FUNCTION "Take-up unit" : VOID	// FC 7
TITLE = TAKE-UP UNIT FUNCTION
AUTHOR : Milesi
VERSION : 0.1
VAR_TEMP
  Min_diameter : REAL ;
  T_up_linear_speed : REAL ;
  T_up_speed_ref : REAL ;
  Take_up_speed_ref : REAL ;
END_VAR
BEGIN
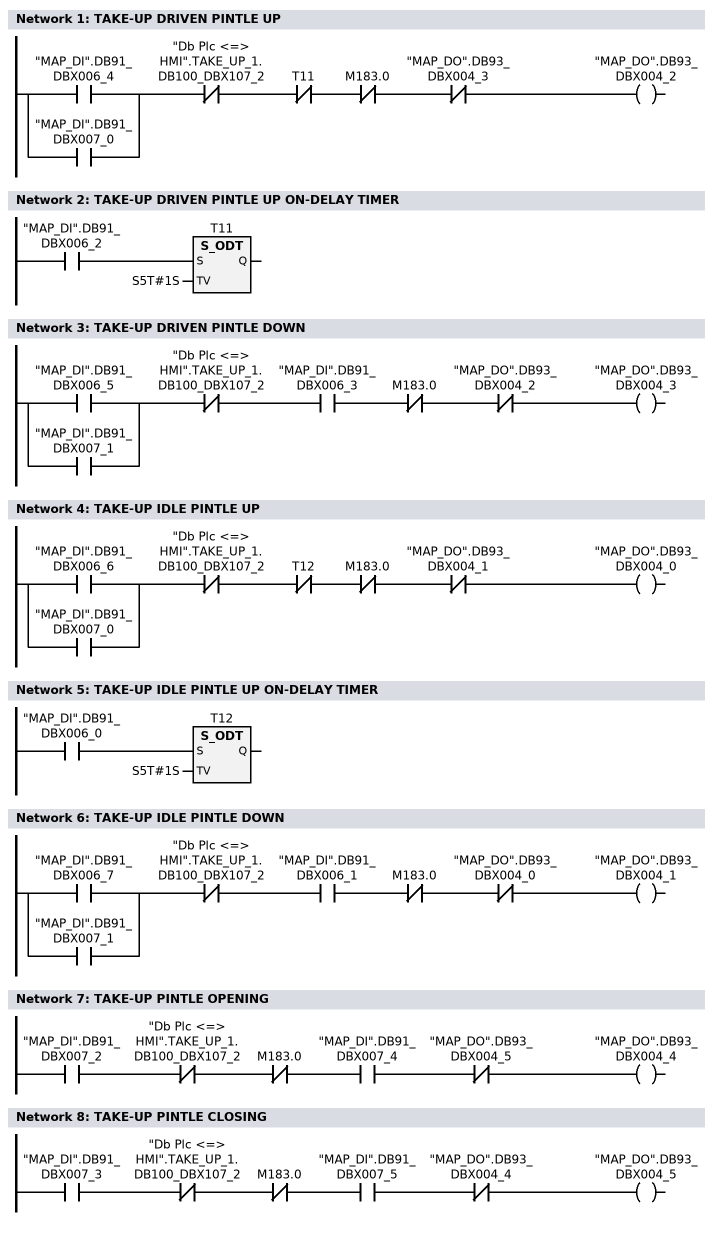
NETWORK
TITLE = TAKE-UP DRIVEN PINTLE UP
      A(;
      O     "MAP_DI".DB91_DBX006_4;
      O     "MAP_DI".DB91_DBX007_0;
      );
      AN    "Db Plc <=> HMI".TAKE_UP_1.DB100_DBX107_2;
      AN    "T11";
      AN    "M183.0";
      AN    "MAP_DO".DB93_DBX004_3;
      =     "MAP_DO".DB93_DBX004_2;
NETWORK
TITLE = TAKE-UP DRIVEN PINTLE UP ON-DELAY TIMER
      A     "MAP_DI".DB91_DBX006_2;
      L     S5T#1S;
      SD    "T11";
      NOP   0;
      NOP   0;
      NOP   0;
      NOP   0;
NETWORK
TITLE = TAKE-UP DRIVEN PINTLE DOWN
      A(;
      O     "MAP_DI".DB91_DBX006_5;
      O     "MAP_DI".DB91_DBX007_1;
      );
      AN    "Db Plc <=> HMI".TAKE_UP_1.DB100_DBX107_2;
      A     "MAP_DI".DB91_DBX006_3;
      AN    "M183.0";
      AN    "MAP_DO".DB93_DBX004_2;
      =     "MAP_DO".DB93_DBX004_3;
NETWORK
TITLE = TAKE-UP IDLE PINTLE UP
      A(;
      O     "MAP_DI".DB91_DBX006_6;
      O     "MAP_DI".DB91_DBX007_0;
      );
      AN    "Db Plc <=> HMI".TAKE_UP_1.DB100_DBX107_2;
      AN    "T12";
      AN    "M183.0";
      AN    "MAP_DO".DB93_DBX004_1;
      =     "MAP_DO".DB93_DBX004_0;
NETWORK
TITLE = TAKE-UP IDLE PINTLE UP ON-DELAY TIMER
      A     "MAP_DI".DB91_DBX006_0;
      L     S5T#1S;
      SD    "T12";
      NOP   0;
      NOP   0;
      NOP   0;
      NOP   0;
NETWORK
TITLE = TAKE-UP IDLE PINTLE DOWN
      A(;
      O     "MAP_DI".DB91_DBX006_7;
      O     "MAP_DI".DB91_DBX007_1;
      );
      AN    "Db Plc <=> HMI".TAKE_UP_1.DB100_DBX107_2;
      A     "MAP_DI".DB91_DBX006_1;
      AN    "M183.0";
      AN    "MAP_DO".DB93_DBX004_0;
      =     "MAP_DO".DB93_DBX004_1;
NETWORK
TITLE = TAKE-UP PINTLE OPENING
      A     "MAP_DI".DB91_DBX007_2;
      AN    "Db Plc <=> HMI".TAKE_UP_1.DB100_DBX107_2;
      AN    "M183.0";
      A     "MAP_DI".DB91_DBX007_4;
      AN    "MAP_DO".DB93_DBX004_5;
      =     "MAP_DO".DB93_DBX004_4;
NETWORK
TITLE = TAKE-UP PINTLE CLOSING
      A     "MAP_DI".DB91_DBX007_3;
      AN    "Db Plc <=> HMI".TAKE_UP_1.DB100_DBX107_2;
      AN    "M183.0";
      A     "MAP_DI".DB91_DBX007_5;
      AN    "MAP_DO".DB93_DBX004_4;
      =     "MAP_DO".DB93_DBX004_5;
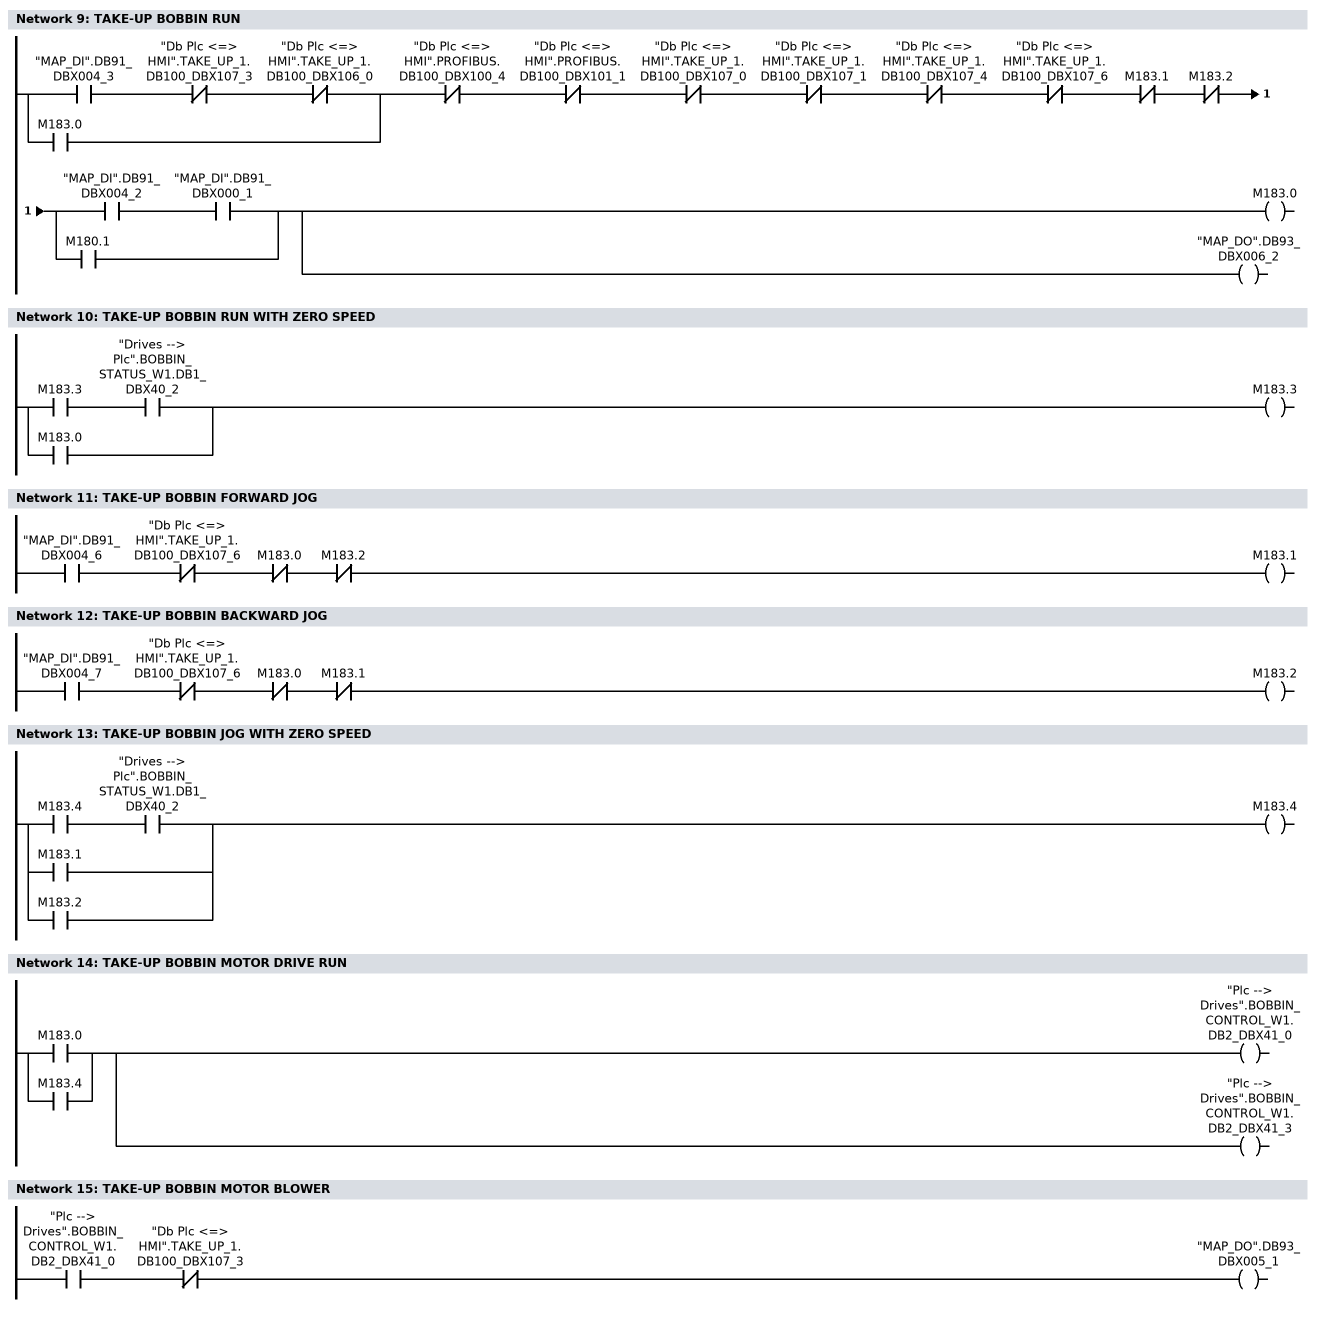
NETWORK
TITLE = TAKE-UP BOBBIN RUN
      A(;
      A     "MAP_DI".DB91_DBX004_3;
      AN    "Db Plc <=> HMI".TAKE_UP_1.DB100_DBX107_3;
      AN    "Db Plc <=> HMI".TAKE_UP_1.DB100_DBX106_0;
      O     "M183.0";
      );
      AN    "Db Plc <=> HMI".PROFIBUS.DB100_DBX100_4;
      AN    "Db Plc <=> HMI".PROFIBUS.DB100_DBX101_1;
      AN    "Db Plc <=> HMI".TAKE_UP_1.DB100_DBX107_0;
      AN    "Db Plc <=> HMI".TAKE_UP_1.DB100_DBX107_1;
      AN    "Db Plc <=> HMI".TAKE_UP_1.DB100_DBX107_4;
      AN    "Db Plc <=> HMI".TAKE_UP_1.DB100_DBX107_6;
      AN    "M183.1";
      AN    "M183.2";
      A(;
      A     "MAP_DI".DB91_DBX004_2;
      A     "MAP_DI".DB91_DBX000_1;
      O     "M180.1";
      );
      =     "M183.0";
      =     "MAP_DO".DB93_DBX006_2;
NETWORK
TITLE = TAKE-UP BOBBIN RUN WITH ZERO SPEED
      A     "M183.3";
      A     "Drives --> Plc".BOBBIN_STATUS_W1.DB1_DBX40_2;
      O     "M183.0";
      =     "M183.3";
NETWORK
TITLE = TAKE-UP BOBBIN FORWARD JOG
      A     "MAP_DI".DB91_DBX004_6;
      AN    "Db Plc <=> HMI".TAKE_UP_1.DB100_DBX107_6;
      AN    "M183.0";
      AN    "M183.2";
      =     "M183.1";
NETWORK
TITLE = TAKE-UP BOBBIN BACKWARD JOG
      A     "MAP_DI".DB91_DBX004_7;
      AN    "Db Plc <=> HMI".TAKE_UP_1.DB100_DBX107_6;
      AN    "M183.0";
      AN    "M183.1";
      =     "M183.2";
NETWORK
TITLE = TAKE-UP BOBBIN JOG WITH ZERO SPEED
      A     "M183.4";
      A     "Drives --> Plc".BOBBIN_STATUS_W1.DB1_DBX40_2;
      O     "M183.1";
      O     "M183.2";
      =     "M183.4";
NETWORK
TITLE = TAKE-UP BOBBIN MOTOR DRIVE RUN
      O     "M183.0";
      O     "M183.4";
      =     "Plc --> Drives".BOBBIN_CONTROL_W1.DB2_DBX41_0;
      =     "Plc --> Drives".BOBBIN_CONTROL_W1.DB2_DBX41_3;
NETWORK
TITLE = TAKE-UP BOBBIN MOTOR BLOWER
      A     "Plc --> Drives".BOBBIN_CONTROL_W1.DB2_DBX41_0;
      AN    "Db Plc <=> HMI".TAKE_UP_1.DB100_DBX107_3;
      =     "MAP_DO".DB93_DBX005_1;
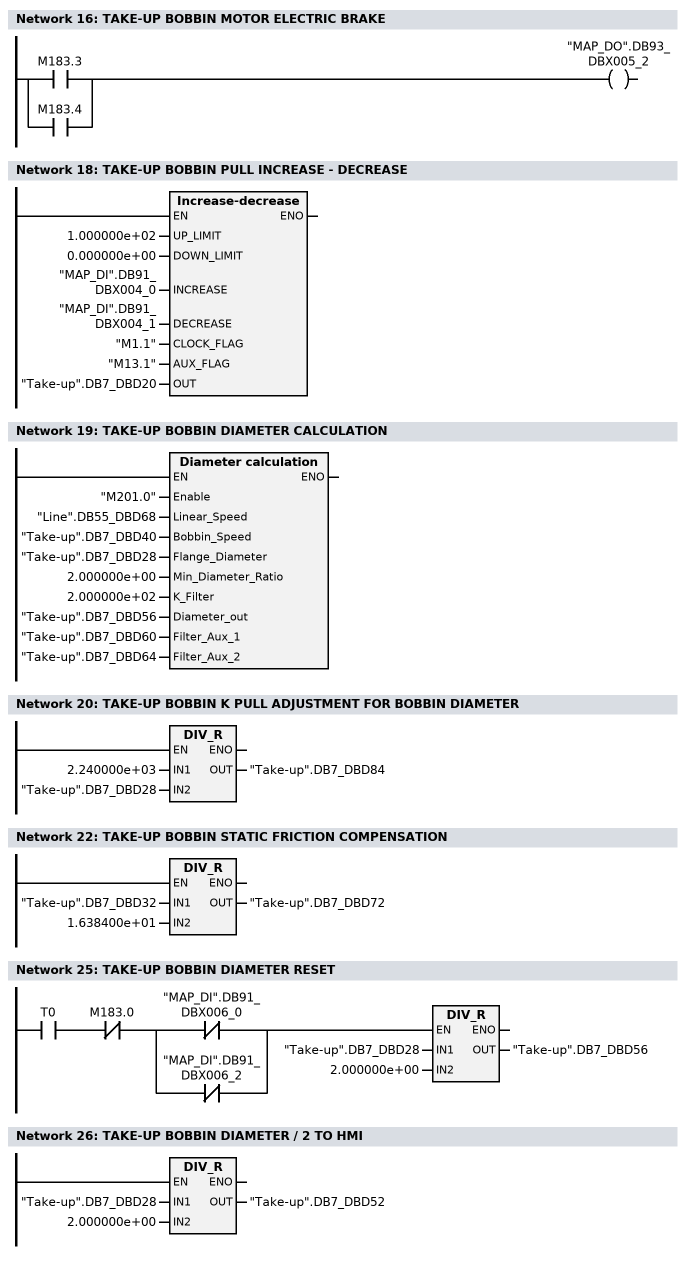
NETWORK
TITLE = TAKE-UP BOBBIN MOTOR ELECTRIC BRAKE
      O     "M183.3";
      O     "M183.4";
      =     "MAP_DO".DB93_DBX005_2;
NETWORK
TITLE = TAKE-UP BOBBIN RPM
      L     "Drives --> Plc".DB1_DBW46;
      ITD;
      DTR;
      L     1.638400e+04;
      /R;
      L     3.031000e+01;
      *R;
      ABS;
      T     "Take-up".DB7_DBD40;
NETWORK
TITLE = TAKE-UP BOBBIN PULL INCREASE - DECREASE
      CALL  "Increase-decrease" (
           UP_LIMIT                 := 1.000000e+02,
           DOWN_LIMIT               := 0.000000e+00,
           INCREASE                 := "MAP_DI".DB91_DBX004_0,
           DECREASE                 := "MAP_DI".DB91_DBX004_1,
           CLOCK_FLAG               := "M1.1",
           AUX_FLAG                 := "M13.1",
           OUT                      := "Take-up".DB7_DBD20);
NETWORK
TITLE = TAKE-UP BOBBIN DIAMETER CALCULATION
      CALL  "Diameter calculation" (
           Enable                   := "M201.0",
           Linear_Speed             := "Line".DB55_DBD68,
           Bobbin_Speed             := "Take-up".DB7_DBD40,
           Flange_Diameter          := "Take-up".DB7_DBD28,
           Min_Diameter_Ratio       := 2.000000e+00,
           K_Filter                 := 2.000000e+02,
           Diameter_out             := "Take-up".DB7_DBD56,
           Filter_Aux_1             := "Take-up".DB7_DBD60,
           Filter_Aux_2             := "Take-up".DB7_DBD64);
NETWORK
TITLE = TAKE-UP BOBBIN K PULL ADJUSTMENT FOR BOBBIN DIAMETER 
      L     2.240000e+03;
      L     "Take-up".DB7_DBD28;
      /R;
      T     "Take-up".DB7_DBD84;
NETWORK
TITLE = TAKE-UP BOBBIN PULL REFERENCE
//Max diameter bobbin = 2240
//Max pull set = 100
//
//(Max diameter bobbin * Max pull set)
//------------------------------------ = 16384
//                 K
//
//    (Max diameter bobbin * Max pull set)   2240 * 100
//K = ------------------------------------ = ---------- = 13.67187
//                    16384                    16384
      L     "Take-up".DB7_DBD56;
      L     "Take-up".DB7_DBD20;
      *R;
      L     1.367187e+01;
      /R;
      L     "Take-up".DB7_DBD84;
      *R;
      L     "Take-up".DB7_DBD72;
      +R;
      L     "Take-up".DB7_DBD76;
      +R;
      T     "Take-up".DB7_DBD68;
NETWORK
TITLE = TAKE-UP BOBBIN STATIC FRICTION COMPENSATION
      L     "Take-up".DB7_DBD32;
      L     1.638400e+01;
      /R;
      T     "Take-up".DB7_DBD72;
NETWORK
TITLE = TAKE-UP BOBBIN DYNAMIC FRICTION COMPENSATION
//Max Bobbin rpm = 30.31
//Max dynamic friction set = 100
//
//(Max Bobbin rpm * Max dynamic friction set) * K = 1638
//
//              1638                                   1638 
//K = ------------------------------------------- = ----------- = 0.54041
//    (Max Bobbin rpm * Max dynamic friction set)   30.31 * 100
      L     "Take-up".DB7_DBD40;
      L     "Take-up".DB7_DBD36;
      *R;
      L     5.404100e-01;
      /R;
      T     "Take-up".DB7_DBD76;
NETWORK
TITLE = TAKE-UP BOBBIN MINIMUM PULL WITH LINE STOP
      A     "M180.1";
      JC    _032;
      L     "Take-up".DB7_DBD56;
      L     "Take-up".DB7_DBD20;
      *R;
      L     1.367187e+01;
      /R;
      L     "Take-up".DB7_DBD24;
      *R;
      L     1.000000e+02;
      /R;
      L     "Take-up".DB7_DBD72;
      +R;
      T     "Take-up".DB7_DBD68;
_032: NOP   0;
NETWORK
TITLE = TAKE-UP BOBBIN DIAMETER RESET
      A     "T0";
      AN    "M183.0";
      A(;
      ON    "MAP_DI".DB91_DBX006_0;
      ON    "MAP_DI".DB91_DBX006_2;
      );
      JNB   _001;
      L     "Take-up".DB7_DBD28;
      L     2.000000e+00;
      /R;
      T     "Take-up".DB7_DBD56;
_001: NOP   0;
NETWORK
TITLE = TAKE-UP BOBBIN DIAMETER / 2 TO HMI
      L     "Take-up".DB7_DBD28;
      L     2.000000e+00;
      /R;
      T     "Take-up".DB7_DBD52;
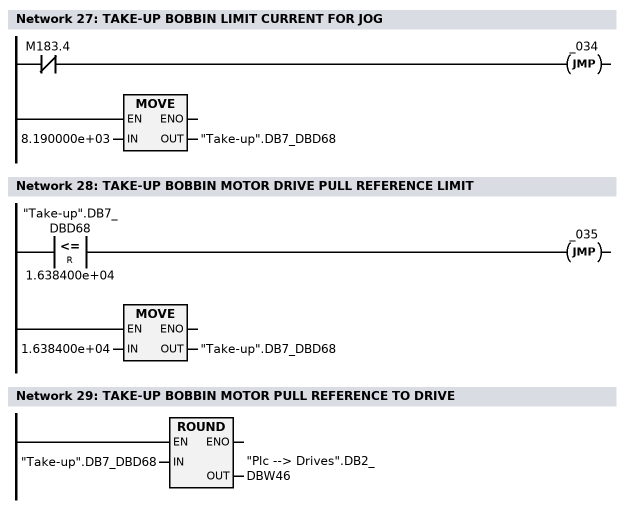
NETWORK
TITLE = TAKE-UP BOBBIN LIMIT CURRENT FOR JOG
      AN    "M183.4";
      JC    _034;
      L     8.190000e+03;
      T     "Take-up".DB7_DBD68;
_034: NOP   0;
NETWORK
TITLE = TAKE-UP BOBBIN MOTOR DRIVE PULL REFERENCE LIMIT
      A(;
      L     "Take-up".DB7_DBD68;
      L     1.638400e+04;
      <=R;
      );
      JC    _035;
      L     1.638400e+04;
      T     "Take-up".DB7_DBD68;
_035: NOP   0;
NETWORK
TITLE = TAKE-UP BOBBIN MOTOR PULL REFERENCE TO DRIVE
      L     "Take-up".DB7_DBD68;
      RND;
      T     "Plc --> Drives".DB2_DBW46;
NETWORK
TITLE = TAKE-UP BOBBIN MOTOR SPEED REFERENCE TO DRIVE
// (network holds code this reader does not know; not shown)
NETWORK
TITLE = TAKE-UP BOBBIN MOTOR RPM TO HMI
      L     "Drives --> Plc".DB1_DBW46;
      ITD;
      DTR;
      L     1.638400e+04;
      /R;
      L     1.515000e+03;
      *R;
      T     "Take-up".DB7_DBD188;
NETWORK
TITLE = TAKE-UP BOBBIN MOTOR CURRENT TO HMI
      L     "Drives --> Plc".DB1_DBW48;
      ITD;
      DTR;
      L     1.638400e+04;
      /R;
      L     2.150000e+01;
      *R;
      T     "Take-up".DB7_DBD192;
NETWORK
TITLE = TAKE-UP BOBBIN MOTOR VOLTAGE TO HMI
      L     "Drives --> Plc".DB1_DBW50;
      ITD;
      DTR;
      L     1.638400e+04;
      /R;
      L     4.000000e+02;
      *R;
      T     "Take-up".DB7_DBD196;
END_FUNCTION

FUNCTION "Capstan alarms" : VOID	// FC 8
TITLE = CAPSTAN ALARMS FUNCTION
AUTHOR : Milesi
VERSION : 0.1
BEGIN
NETWORK
TITLE = CAPSTAN MOTOR DRIVE PROFIBUS SLAVE 5 FAULT
      A(;
      L     "MB304";
      L     5;
      ==I;
      );
      AN    "M300.5";
      S     "Db Plc <=> HMI".PROFIBUS.DB100_DBX101_2;
NETWORK
TITLE = CAPSTAN MOTOR DRIVE FAULT
      A     "T0";
      A     "Drives --> Plc".CAPSTAN_STATUS_W1.DB1_DBX81_3;
      S     "Db Plc <=> HMI".CAPSTAN.DB100_DBX109_6;
NETWORK
TITLE = CAPSTAN MOTOR OVERTEMPERATURE
      A     "T0";
      A     "Drives --> Plc".CAPSTAN_STATUS_W2.DB1_DBX82_1;
      S     "Db Plc <=> HMI".CAPSTAN.DB100_DBX109_7;
NETWORK
TITLE = CAPSTAN MOTOR BLOWER OVERLOAD
      A     "T0";
      A     "MAP_DI".DB91_DBX012_0;
      =     "Db Plc <=> HMI".CAPSTAN.DB100_DBX109_0;
NETWORK
TITLE = CAPSTAN MOTOR BRAKE CONTROL
      A     "T0";
      A     "M180.1";
      AN    "MAP_DI".DB91_DBX012_2;
      A     "T2";
      S     "Db Plc <=> HMI".CAPSTAN.DB100_DBX109_2;
NETWORK
TITLE = CAPSTAN MAIN AIR MINIMUM PRESSURE
      A     "T0";
      A     "M180.1";
      AN    "MAP_DI".DB91_DBX012_1;
      S     "M170.1";
NETWORK
TITLE =
      A     "T0";
      A(;
      ON    "MAP_DI".DB91_DBX012_1;
      O     "M170.1";
      );
      =     "Db Plc <=> HMI".CAPSTAN.DB100_DBX109_3;
NETWORK
TITLE = CABLE BLOCK OPEN
      A     "T0";
      AN    "M180.1";
      A     "M21.1";
      AN    "M184.0";
      AN    "M184.1";
      A     "MAP_DI".DB91_DBX012_3;
      =     "Db Plc <=> HMI".CAPSTAN.DB100_DBX109_4;
NETWORK
TITLE = CABLE BLOCK CLOSE AFTER RUN
      A     "T0";
      A(;
      O     "M180.1";
      O     "M21.3";
      O     "M184.0";
      O     "M184.1";
      );
      AN    "MAP_DI".DB91_DBX012_3;
      A     "T2";
      S     "Db Plc <=> HMI".CAPSTAN.DB100_DBX109_5;
NETWORK
TITLE = CAPSTAN GENERAL ALARM 
      AN    "Db Plc <=> HMI".PROFIBUS.DB100_DBX101_2;
      AN    "Db Plc <=> HMI".CAPSTAN.DB100_DBX109_0;
      AN    "Db Plc <=> HMI".CAPSTAN.DB100_DBX109_2;
      AN    "Db Plc <=> HMI".CAPSTAN.DB100_DBX109_3;
      AN    "Db Plc <=> HMI".CAPSTAN.DB100_DBX109_4;
      AN    "Db Plc <=> HMI".CAPSTAN.DB100_DBX109_5;
      AN    "Db Plc <=> HMI".CAPSTAN.DB100_DBX109_6;
      AN    "Db Plc <=> HMI".CAPSTAN.DB100_DBX109_7;
      =     "M197.3";
END_FUNCTION

FUNCTION "Capstan unit" : VOID	// FC 9
TITLE = CAPSTAN UNIT FUNCTION
AUTHOR : Milesi
VERSION : 0.1
VAR_TEMP
  Cable_diameter_K : REAL ;
END_VAR
BEGIN
NETWORK
TITLE = CAPSTAN FORWARD JOG
      A     "MAP_DI".DB91_DBX012_5;
      AN    "Db Plc <=> HMI".CAPSTAN.DB100_DBX109_0;
      AN    "Db Plc <=> HMI".CAPSTAN.DB100_DBX109_2;
      AN    "Db Plc <=> HMI".CAPSTAN.DB100_DBX109_5;
      AN    "Db Plc <=> HMI".CAPSTAN.DB100_DBX109_6;
      AN    "Db Plc <=> HMI".CAPSTAN.DB100_DBX109_7;
      AN    "M180.1";
      AN    "M184.1";
      =     "M184.0";
NETWORK
TITLE = CAPSTAN BACKWARD JOG
      A     "MAP_DI".DB91_DBX012_6;
      AN    "Db Plc <=> HMI".CAPSTAN.DB100_DBX109_0;
      AN    "Db Plc <=> HMI".CAPSTAN.DB100_DBX109_2;
      AN    "Db Plc <=> HMI".CAPSTAN.DB100_DBX109_5;
      AN    "Db Plc <=> HMI".CAPSTAN.DB100_DBX109_6;
      AN    "Db Plc <=> HMI".CAPSTAN.DB100_DBX109_7;
      AN    "M180.1";
      AN    "M184.0";
      =     "M184.1";
NETWORK
TITLE = CAPSTAN JOG WITH ZERO SPEED
      A     "M184.2";
      A     "Drives --> Plc".CAPSTAN_STATUS_W1.DB1_DBX80_2;
      O     "M184.0";
      O     "M184.1";
      =     "M184.2";
NETWORK
TITLE = CAPSTAN MOTOR DRIVE RUN
      O     "M21.3";
      O     "M180.1";
      O     "M184.2";
      =     "Plc --> Drives".CAPSTAN_CONTROL_W1.DB2_DBX81_0;
      =     "Plc --> Drives".CAPSTAN_CONTROL_W1.DB2_DBX81_3;
NETWORK
TITLE = CAPSTAN MOTOR BLOWER
      A     "Plc --> Drives".CAPSTAN_CONTROL_W1.DB2_DBX81_0;
      AN    "Db Plc <=> HMI".CAPSTAN.DB100_DBX109_0;
      =     "MAP_DO".DB93_DBX001_2;
NETWORK
TITLE = CAPSTAN BRAKE BLOCK
      A     "M21.1";
      AN    "M180.1";
      AN    "M184.2";
      =     "MAP_DO".DB93_DBX001_3;
NETWORK
TITLE = CAPSTAN CABLE BLOCK
      O     "M180.1";
      O     "M21.3";
      O     "M184.2";
      O;
      A     "MAP_DI".DB91_DBX012_4;
      AN    "M180.1";
      A     "M21.1";
      AN    "M184.2";
      =     "MAP_DO".DB93_DBX001_4;
NETWORK
TITLE = CABLE DIAMETER CONSTANT
//             Capstan pulley Ш + Cable Ш
//K (Cable Ш)= --------------------------
//                 Capstan pulley Ш
      L     2.500000e+03;
      L     "Line".DB55_DBD56;
      +R;
      L     2.500000e+03;
      /R;
      T     #Cable_diameter_K;
NETWORK
TITLE = CAPSTAN MOTOR DRIVE SPEED REFERENCE
// (network holds code this reader does not know; not shown)
NETWORK
TITLE = CAPSTAN MOTOR RPM TO HMI
      L     "Drives --> Plc".DB1_DBW86;
      ITD;
      DTR;
      L     1.638400e+04;
      /R;
      L     1.873000e+03;
      *R;
      T     "Capstan".DB9_DBD188;
NETWORK
TITLE = CAPSTAN MOTOR CURRENT TO HMI
      L     "Drives --> Plc".DB1_DBW88;
      ITD;
      DTR;
      L     1.638400e+04;
      /R;
      L     2.800000e+02;
      *R;
      T     "Capstan".DB9_DBD192;
NETWORK
TITLE = CAPSTAN MOTOR VOLTAGE TO HMI
      L     "Drives --> Plc".DB1_DBW90;
      ITD;
      DTR;
      L     1.638400e+04;
      /R;
      L     4.000000e+02;
      *R;
      T     "Capstan".DB9_DBD196;
END_FUNCTION

FUNCTION "Door Cage Lock" : VOID	// FC 10
VERSION : 0.1
VAR_INPUT
  Door_Open : BOOL ;
  Button_Door_Up : BOOL ;
  Button_Door_Down : BOOL ;
END_VAR
VAR_OUTPUT
  Door_Lock : BOOL ;
  Door_UnLock : BOOL ;
END_VAR
VAR_TEMP
  Release_Door_Lock : BOOL ;
END_VAR
BEGIN
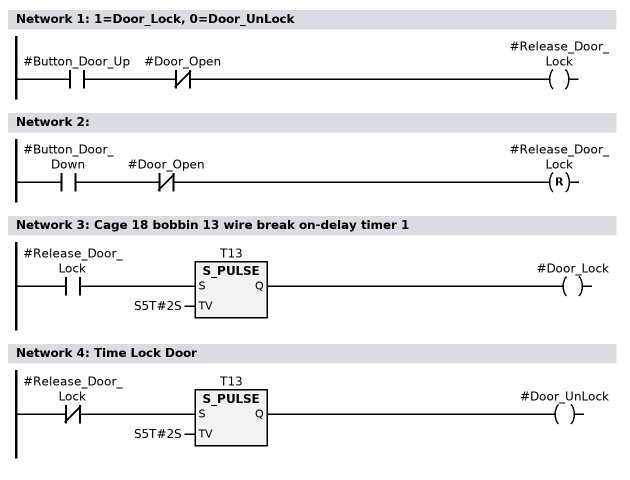
NETWORK
TITLE = 1=Door_Lock, 0=Door_UnLock
      A     #Button_Door_Up;
      AN    #Door_Open;
      =     #Release_Door_Lock;
NETWORK
TITLE =
      A     #Button_Door_Down;
      AN    #Door_Open;
      R     #Release_Door_Lock;
NETWORK
TITLE = Cage 18 bobbin 13 wire break on-delay timer 1
      A     #Release_Door_Lock;
      L     S5T#2S;
      SP    "T13";
      NOP   0;
      NOP   0;
      NOP   0;
      A     "T13";
      =     #Door_Lock;
NETWORK
TITLE = Time Lock Door
      AN    #Release_Door_Lock;
      L     S5T#2S;
      SP    "T13";
      NOP   0;
      NOP   0;
      NOP   0;
      A     "T13";
      =     #Door_UnLock;
END_FUNCTION

FUNCTION "Cage common function" : VOID	// FC 13
TITLE = CAGES COMMON FUNCTION
AUTHOR : Milesi
VERSION : 0.1
BEGIN
NETWORK
TITLE = LOADING RUN FROM ONE O MORE CAGES
      O     "M181.2";
      O     "M181.3";
      O     "M181.4";
      O     "M181.5";
      =     "M20.0";
NETWORK
TITLE = LINE JOG OF ONE O MORE CAGE
      O     "MAP_DI".DB91_DBX022_1;
      O     "MAP_DI".DB91_DBX042_1;
      O     "MAP_DI".DB91_DBX062_1;
      O     "MAP_DI".DB91_DBX082_1;
      =     "M20.2";
NETWORK
TITLE = LOADING RUN PUSH-BUTTON OF ONE O MORE CAGE 
      O     "MAP_DI".DB91_DBX022_2;
      O     "MAP_DI".DB91_DBX042_2;
      O     "MAP_DI".DB91_DBX062_2;
      O     "MAP_DI".DB91_DBX082_2;
      =     "M20.3";
NETWORK
TITLE = PREFORMING LINE JOG OF ONE O MORE CAGE
      O     "MAP_DI".DB91_DBX085_1;
      O     "MAP_DI".DB91_DBX065_1;
      O     "MAP_DI".DB91_DBX045_1;
      O     "MAP_DI".DB91_DBX025_1;
      =     "M20.4";
NETWORK
TITLE = LOADING RUN FROM ONE OF CAGE WITH PISTON DISENGAGED
      O     "M180.4";
      O     "M180.5";
      O     "M180.6";
      O     "M180.7";
      =     "M20.6";
NETWORK
TITLE = PREFORMING LINE STOP GLOBAL PUSH-BUTTONS
      A     "MAP_DI".DB91_DBX085_0;
      A     "MAP_DI".DB91_DBX065_0;
      A     "MAP_DI".DB91_DBX045_0;
      A     "MAP_DI".DB91_DBX025_0;
      =     "M20.7";
NETWORK
TITLE = LINE STOP GLOBAL PUSH-BUTTONS
      A     "MAP_DI".DB91_DBX002_0;
      A     "MAP_DI".DB91_DBX099_3;
      A     "MAP_DI".DB91_DBX082_0;
      A     "MAP_DI".DB91_DBX062_0;
      A     "MAP_DI".DB91_DBX042_0;
      A     "MAP_DI".DB91_DBX022_0;
      =     "M21.0";
NETWORK
TITLE = NOT LOADING RUN FROM ALL CAGE
      A(;
      ON    "M180.4";
      ON    "M190.0";
      );
      A(;
      ON    "M180.5";
      ON    "M188.0";
      );
      A(;
      ON    "M180.6";
      ON    "M186.0";
      );
      A(;
      ON    "M180.7";
      ON    "M192.0";
      );
      =     "M21.1";
NETWORK
TITLE = LOADING RUN FROM ONE OF CAGE ON WITH PISTON DISENGAGED
      A     "M180.4";
      A     "M190.0";
      O;
      A     "M180.5";
      A     "M188.0";
      O;
      A     "M180.6";
      A     "M186.0";
      O;
      A     "M180.7";
      A     "M192.0";
      =     "M21.3";
END_FUNCTION

FUNCTION "Cage 24 alarms" : VOID	// FC 14
TITLE = CAGE 24 ALARMS FUNCTION
AUTHOR : Milesi
VERSION : 0.1
VAR_TEMP
  T4_time : WORD ;
END_VAR
BEGIN
NETWORK
TITLE = CAGE 24 MOTOR DRIVE PROFIBUS SLAVE 7 FAULT
      A(;
      L     "MB304";
      L     7;
      ==I;
      );
      AN    "M300.5";
      S     "Db Plc <=> HMI".PROFIBUS.DB100_DBX101_6;
NETWORK
TITLE = CAGE 24 ET200M PROFIBUS SLAVE 21 FAULT
      A(;
      L     "MB304";
      L     21;
      ==I;
      );
      AN    "M300.5";
      S     "Db Plc <=> HMI".PROFIBUS.DB100_DBX100_5;
NETWORK
TITLE = CAGE 24 OPEN FRONT GUARD
      A     "T0";
      A     "M180.1";
      AN    "MAP_DI".DB91_DBX021_6;
      A     "M192.0";
      S     "M171.4";
NETWORK
TITLE =
      A     "T0";
      A(;
      ON    "MAP_DI".DB91_DBX021_6;
      O     "M171.4";
      );
      A     "M192.0";
      =     "Db Plc <=> HMI".CAGE24_1.DB100_DBX112_00;
NETWORK
TITLE = CAGE 24 PRESENCE OF MAN
      A     "T0";
      AN    "MAP_DI".DB91_DBX021_7;
      AN    "M180.1";
      A     "M192.0";
      =     "Db Plc <=> HMI".CAGE24_1.DB100_DBX112_01;
NETWORK
TITLE = CAGE 24 LOADING ENGAGED
      A     "T0";
      A     "MAP_DI".DB91_DBX020_5;
      AN    "MAP_DI".DB91_DBX020_6;
      A     "M017.2";
      =     "Db Plc <=> HMI".CAGE24_1.DB100_DBX112_02;
NETWORK
TITLE = CAGE 24 LOADING GEAR BOX NOT ENGAGED
      A     "T0";
      AN    "MAP_DI".DB91_DBX020_5;
      AN    "MAP_DI".DB91_DBX020_6;
      =     "Db Plc <=> HMI".CAGE24_1.DB100_DBX112_03;
NETWORK
TITLE = CAGE 24 LOADING MOTOR OVERLOAD
      A     "T0";
      A     "MAP_DI".DB91_DBX018_2;
      =     "Db Plc <=> HMI".CAGE24_1.DB100_DBX112_04;
NETWORK
TITLE = CAGE 24 AIR PIPE NOT IN POSITION
      A     "T0";
      A     "M180.1";
      AN    "MAP_DI".DB91_DBX020_7;
      A     "M192.0";
      S     "M170.2";
NETWORK
TITLE =
      A     "T0";
      A(;
      ON    "MAP_DI".DB91_DBX020_7;
      O     "M170.2";
      );
      =     "Db Plc <=> HMI".CAGE24_1.DB100_DBX112_05;
NETWORK
TITLE = CAGE 24 PISTON INSIDE CAGE
      A     "T0";
      A     "M180.1";
      AN    "MAP_DI".DB91_DBX020_4;
      A     "M192.0";
      S     "M170.3";
NETWORK
TITLE =
      A     "T0";
      A(;
      ON    "MAP_DI".DB91_DBX020_4;
      O     "M170.3";
      );
      =     "Db Plc <=> HMI".CAGE24_1.DB100_DBX112_07;
NETWORK
TITLE = CAGE 24 24VDC POWER SUPPLY OVERLOAD
      A     "T0";
      AN    "MAP_DI".DB91_DBX018_1;
      =     "Db Plc <=> HMI".CAGE24_1.DB100_DBX113_00;
NETWORK
TITLE = CAGE 24 230VAC POWER SUPPLY OVERLOAD
      A     "T0";
      AN    "MAP_DI".DB91_DBX018_0;
      =     "Db Plc <=> HMI".CAGE24_1.DB100_DBX113_01;
NETWORK
TITLE = CAGE 24 MOTOR BLOWER OVERLOAD
      A     "T0";
      A     "MAP_DI".DB91_DBX018_3;
      =     "Db Plc <=> HMI".CAGE24_1.DB100_DBX113_02;
NETWORK
TITLE = CAGE 24 LOADING PLATFORM MOTOR OVERLOAD
NETWORK
TITLE = CAGE 24 GUARD BLOWER MOTOR OVERLOAD
      A     "T0";
      A     "MAP_DI".DB91_DBX018_7;
      =     "Db Plc <=> HMI".CAGE24_1.DB100_DBX113_05;
NETWORK
TITLE = CAGE 24 OPEN FRONT DOOR
//      U(    
//      U(    
//      U     T      0
//      U     M    178.0
//      O     M    180.1
//      O     M     21.3
//      )     
//      L     S5T#2S
//      SE    T     19
//      NOP   0
//      NOP   0
//      NOP   0
//      U     T     19
//      )     
//      UN    DB91.DBX   21.3
//      U     M    192.0
//      S     DB100.DBX  113.6
NETWORK
TITLE = CAGE 24 OPEN REAR DOORS
      A     "T0";
      A     "M180.1";
      AN    "MAP_DI".DB91_DBX021_4;
      A     "M192.0";
      S     "M172.1";
NETWORK
TITLE =
      A     "T0";
      A(;
      ON    "MAP_DI".DB91_DBX021_4;
      O     "M172.1";
      );
      A     "M192.0";
      =     "Db Plc <=> HMI".CAGE24_1.DB100_DBX113_07;
NETWORK
TITLE = CAGE 18 BREAK WIRE FROM RING 
      A     "T0";
      A     "T1";
      AN    "MAP_DI".DB91_DBX021_2;
      A     "M192.0";
      S     "Db Plc <=> HMI".CAGE24_3.DB100_DBX117_06;
NETWORK
TITLE = CAGE 24 MAIN AIR MINIMUM PRESSURE
      A     "T0";
      A     "M180.1";
      AN    "MAP_DI".DB91_DBX020_2;
      A     "M192.0";
      S     "M172.2";
NETWORK
TITLE =
      A     "T0";
      A(;
      ON    "MAP_DI".DB91_DBX020_2;
      O     "M172.2";
      );
      =     "Db Plc <=> HMI".CAGE24_4.DB100_DBX118_00;
NETWORK
TITLE = CAGE 24 BOBBIN BRAKES AIR TANK MINIMUM PRESSURE
      A     "T0";
      AN    "Db Plc <=> HMI".PROFIBUS.DB100_DBX100_5;
      AN    "MAP_DI".DB91_DBX027_4;
      A     "M192.0";
      S     "Db Plc <=> HMI".CAGE24_4.DB100_DBX118_01;
NETWORK
TITLE = CAGE 24 LINE 1 PINTLES OPEN
      A     "T0";
      A     "M180.1";
      AN    "MAP_DI".DB91_DBX027_5;
      A     "M192.0";
      S     "M170.4";
NETWORK
TITLE =
      A     "T0";
      A(;
      ON    "MAP_DI".DB91_DBX027_5;
      O     "M170.4";
      );
      =     "Db Plc <=> HMI".CAGE24_4.DB100_DBX118_02;
NETWORK
TITLE = CAGE 24 LINE 2 PINTLES OPEN
      A     "T0";
      A     "M180.1";
      AN    "MAP_DI".DB91_DBX027_6;
      A     "M192.0";
      S     "M170.5";
NETWORK
TITLE =
      A     "T0";
      A(;
      ON    "MAP_DI".DB91_DBX027_6;
      O     "M170.5";
      );
      =     "Db Plc <=> HMI".CAGE24_4.DB100_DBX118_03;
NETWORK
TITLE = CAGE 24 LINE 3 PINTLES OPEN
      A     "T0";
      A     "M180.1";
      AN    "MAP_DI".DB91_DBX027_7;
      A     "M192.0";
      S     "M170.6";
NETWORK
TITLE =
      A     "T0";
      A(;
      ON    "MAP_DI".DB91_DBX027_7;
      O     "M170.6";
      );
      =     "Db Plc <=> HMI".CAGE24_4.DB100_DBX118_04;
NETWORK
TITLE = CAGE 24 OPEN PINTLES LAMP
      ON    "MAP_DI".DB91_DBX027_5;
      ON    "MAP_DI".DB91_DBX027_6;
      ON    "MAP_DI".DB91_DBX027_7;
      =     "M179.5";
      =     "MAP_DO".DB93_DBX022_0;
NETWORK
TITLE = CAGE 24 MOTOR DRIVE FAULT
      A     "T0";
      A     "Drives --> Plc".CAGE_24_STATUS_W1.DB1_DBX161_3;
      S     "Db Plc <=> HMI".CAGE24_4.DB100_DBX118_05;
NETWORK
TITLE = CAGE 24 MOTOR OVERTEMPERATURE
      A     "T0";
      A     "Drives --> Plc".CAGE_24_STATUS_W2.DB1_DBX162_1;
      S     "Db Plc <=> HMI".CAGE24_4.DB100_DBX118_06;
NETWORK
TITLE = CAGE 24 OVERSPEED
      A     "T0";
      A     "M180.1";
      A(;
      L     "Cage 24".DB15_DBD108;
      L     2.450000e+02;
      >=R;
      );
      A     "M192.0";
      S     "Db Plc <=> HMI".CAGE24_4.DB100_DBX118_07;
NETWORK
TITLE = CAGE 24 BRAKES CONTROL
      A     "T0";
      A     "T2";
      AN    "MAP_DI".DB91_DBX020_1;
      A     "M192.0";
      S     "Db Plc <=> HMI".CAGE24_4.DB100_DBX119_00;
NETWORK
TITLE = CAGE 24 PLATFORM UP
NETWORK
TITLE = CAGE 24 HIDRAULIC UNIT MINIMUM OIL LEVEL  
NETWORK
TITLE = CAGE 24 GENERAL ALARM
      AN    "Db Plc <=> HMI".PROFIBUS.DB100_DBX100_5;
      AN    "Db Plc <=> HMI".PROFIBUS.DB100_DBX101_6;
      AN    "Db Plc <=> HMI".CAGE24_1.DB100_DBX112_00;
      AN    "Db Plc <=> HMI".CAGE24_1.DB100_DBX112_01;
      AN    "Db Plc <=> HMI".CAGE24_1.DB100_DBX112_03;
      AN    "Db Plc <=> HMI".CAGE24_1.DB100_DBX112_05;
      AN    "Db Plc <=> HMI".CAGE24_1.DB100_DBX112_07;
      AN    "Db Plc <=> HMI".CAGE24_1.DB100_DBX113_00;
      AN    "Db Plc <=> HMI".CAGE24_1.DB100_DBX113_01;
      AN    "Db Plc <=> HMI".CAGE24_1.DB100_DBX113_02;
      AN    "Db Plc <=> HMI".CAGE24_1.DB100_DBX113_06;
      AN    "Db Plc <=> HMI".CAGE24_1.DB100_DBX113_07;
      AN    "Db Plc <=> HMI".CAGE24_2.DB100_DBX114_00;
      AN    "Db Plc <=> HMI".CAGE24_2.DB100_DBX114_01;
      AN    "Db Plc <=> HMI".CAGE24_2.DB100_DBX114_02;
      AN    "Db Plc <=> HMI".CAGE24_2.DB100_DBX114_03;
      AN    "Db Plc <=> HMI".CAGE24_2.DB100_DBX114_04;
      AN    "Db Plc <=> HMI".CAGE24_2.DB100_DBX114_05;
      AN    "Db Plc <=> HMI".CAGE24_2.DB100_DBX114_06;
      AN    "Db Plc <=> HMI".CAGE24_2.DB100_DBX114_07;
      AN    "Db Plc <=> HMI".CAGE24_2.DB100_DBX115_00;
      AN    "Db Plc <=> HMI".CAGE24_2.DB100_DBX115_01;
      AN    "Db Plc <=> HMI".CAGE24_2.DB100_DBX115_02;
      AN    "Db Plc <=> HMI".CAGE24_2.DB100_DBX115_03;
      AN    "Db Plc <=> HMI".CAGE24_2.DB100_DBX115_04;
      AN    "Db Plc <=> HMI".CAGE24_2.DB100_DBX115_05;
      AN    "Db Plc <=> HMI".CAGE24_2.DB100_DBX115_06;
      AN    "Db Plc <=> HMI".CAGE24_2.DB100_DBX115_07;
      AN    "Db Plc <=> HMI".CAGE24_3.DB100_DBX116_00;
      AN    "Db Plc <=> HMI".CAGE24_3.DB100_DBX116_01;
      AN    "Db Plc <=> HMI".CAGE24_3.DB100_DBX116_02;
      AN    "Db Plc <=> HMI".CAGE24_3.DB100_DBX116_03;
      AN    "Db Plc <=> HMI".CAGE24_3.DB100_DBX116_04;
      AN    "Db Plc <=> HMI".CAGE24_3.DB100_DBX116_05;
      AN    "Db Plc <=> HMI".CAGE24_3.DB100_DBX116_06;
      AN    "Db Plc <=> HMI".CAGE24_3.DB100_DBX116_07;
      AN    "Db Plc <=> HMI".CAGE24_3.DB100_DBX117_06;
      AN    "Db Plc <=> HMI".CAGE24_3.DB100_DBX117_07;
      AN    "Db Plc <=> HMI".CAGE24_4.DB100_DBX118_00;
      AN    "Db Plc <=> HMI".CAGE24_4.DB100_DBX118_01;
      AN    "Db Plc <=> HMI".CAGE24_4.DB100_DBX118_02;
      AN    "Db Plc <=> HMI".CAGE24_4.DB100_DBX118_03;
      AN    "Db Plc <=> HMI".CAGE24_4.DB100_DBX118_04;
      AN    "Db Plc <=> HMI".CAGE24_4.DB100_DBX118_05;
      AN    "Db Plc <=> HMI".CAGE24_4.DB100_DBX118_06;
      AN    "Db Plc <=> HMI".CAGE24_4.DB100_DBX118_07;
      AN    "Db Plc <=> HMI".CAGE24_4.DB100_DBX119_00;
      ON    "M192.0";
      =     "M195.3";
END_FUNCTION

FUNCTION "Cage 24 unit" : VOID	// FC 15
TITLE = CAGE 24 UNIT FUNCTION
AUTHOR : Milesi
VERSION : 0.1
VAR_TEMP
  Brake_value : INT ;
END_VAR
BEGIN
NETWORK
TITLE = CAGE 24 OFF
      A(;
      L     "Cage 24".DB15_DBW2;
      L     0;
      ==I;
      );
      AN    "M180.1";
      AN    "M20.0";
      JNB   _001;
      R     "M192.0";
_001: NOP   0;
NETWORK
TITLE = CAGE 24 ON
      A(;
      L     "Cage 24".DB15_DBW2;
      L     1;
      ==I;
      );
      AN    "M180.1";
      AN    "M20.0";
      JNB   _040;
      S     "M192.0";
_040: NOP   0;
NETWORK
TITLE = CAGE 24 Z ROTATION
      A(;
      L     "Cage 24".DB15_DBW4;
      L     0;
      ==I;
      );
      AN    "M180.1";
      AN    "M20.0";
      JNB   _002;
      S     "M192.2";
      R     "M192.3";
_002: NOP   0;
NETWORK
TITLE = CAGE 24 S ROTATION
      A(;
      L     "Cage 24".DB15_DBW4;
      L     1;
      ==I;
      );
      AN    "M180.1";
      AN    "M20.0";
      JNB   _003;
      S     "M192.3";
      R     "M192.2";
_003: NOP   0;
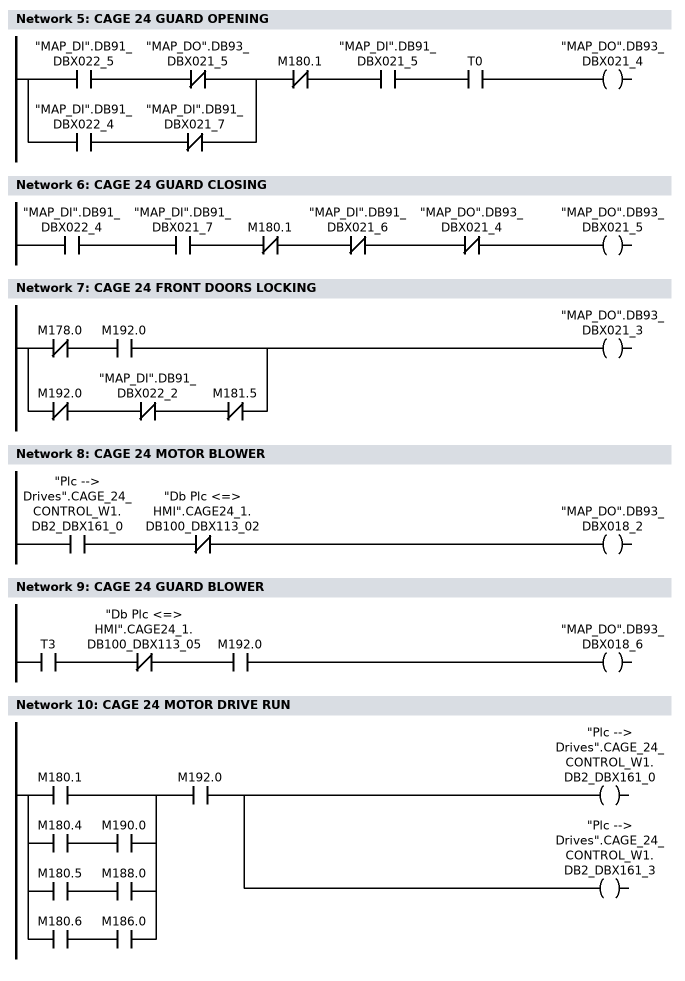
NETWORK
TITLE = CAGE 24 GUARD OPENING
      A(;
      A     "MAP_DI".DB91_DBX022_5;
      AN    "MAP_DO".DB93_DBX021_5;
      O;
      A     "MAP_DI".DB91_DBX022_4;
      AN    "MAP_DI".DB91_DBX021_7;
      );
      AN    "M180.1";
      A     "MAP_DI".DB91_DBX021_5;
      A     "T0";
      =     "MAP_DO".DB93_DBX021_4;
NETWORK
TITLE = CAGE 24 GUARD CLOSING
      A     "MAP_DI".DB91_DBX022_4;
      A     "MAP_DI".DB91_DBX021_7;
//      U     E     46.0
      AN    "M180.1";
      AN    "MAP_DI".DB91_DBX021_6;
      AN    "MAP_DO".DB93_DBX021_4;
      =     "MAP_DO".DB93_DBX021_5;
NETWORK
TITLE = CAGE 24 FRONT DOORS LOCKING
      AN    "M178.0";
      A     "M192.0";
      O;
      AN    "M192.0";
      AN    "MAP_DI".DB91_DBX022_2;
      AN    "M181.5";
      =     "MAP_DO".DB93_DBX021_3;
NETWORK
TITLE = CAGE 24 MOTOR BLOWER 
      A     "Plc --> Drives".CAGE_24_CONTROL_W1.DB2_DBX161_0;
      AN    "Db Plc <=> HMI".CAGE24_1.DB100_DBX113_02;
      =     "MAP_DO".DB93_DBX018_2;
NETWORK
TITLE = CAGE 24 GUARD BLOWER
      A     "T3";
      AN    "Db Plc <=> HMI".CAGE24_1.DB100_DBX113_05;
      A     "M192.0";
      =     "MAP_DO".DB93_DBX018_6;
NETWORK
TITLE = CAGE 24 MOTOR DRIVE RUN
      A(;
      O     "M180.1";
      O;
      A     "M180.4";
      A     "M190.0";
      O;
      A     "M180.5";
      A     "M188.0";
      O;
      A     "M180.6";
      A     "M186.0";
      );
      A     "M192.0";
      =     "Plc --> Drives".CAGE_24_CONTROL_W1.DB2_DBX161_0;
      =     "Plc --> Drives".CAGE_24_CONTROL_W1.DB2_DBX161_3;
NETWORK
TITLE = CAGE 24 LAY SET ENABLE
      O     "M180.1";
      O     "M180.7";
      O(;
      A     "M180.4";
      A     "M190.0";
      );
      O(;
      A     "M180.5";
      A     "M188.0";
      );
      O(;
      A     "M180.6";
      A     "M186.0";
      );
      JC    _lay;
      L     "Cage 24".DB15_DBD20;
      T     "Cage 24".DB15_DBD24;
      JU    end1;
_lay: L     "Cage 24".DB15_DBD24;
      T     "Cage 24".DB15_DBD20;
end1: NOP   0;
NETWORK
TITLE = CAGE 24 MOTOR REFERENCE
//Max Linear Speed = 60 m/min
//Max Cage Rpm = 240
//
//Max Linear Speed              60000
//---------------- = Cage Lay = ----- = 250
//  Max Cage Rpm                 240
//
//                             Max Linear Speed
//Max Cage Rpm = 240 = 16384 = ---------------- * K
//                                Cage Lay
//
//    Cage Lay * 16384    250 * 16384
//K = ---------------- = ------------- = 68266.66
//    Max Linear Speed        60
// (network holds code this reader does not know; not shown)
NETWORK
TITLE = CAGE 24 MAX LINEAR SPEED TO START
      AN    "M200.1";
      JNB   _017;
      L     "Cage 24".DB15_DBD24;
      L     1.550000e-01;
      *R;
      JU    _018;
_017: L     "Cage 24".DB15_DBD24;
      L     2.300000e-01;
      *R;
_018: T     "Cage 24".DB15_DBD120;
      O(;
      L     6.000000e+01;
      >R;
      );
      ON    "M192.0";
      JNB   _014;
      T     "Cage 24".DB15_DBD120;
_014: NOP   0;
NETWORK
TITLE = CAGE 24 MAX LINEAR SPEED
      L     "Cage 24".DB15_DBD24;
      L     2.400000e-01;
      *R;
      T     "Cage 24".DB15_DBD96;
      O(;
      L     6.000000e+01;
      >R;
      );
      ON    "M192.0";
      JNB   _015;
      T     "Cage 24".DB15_DBD96;
_015: NOP   0;
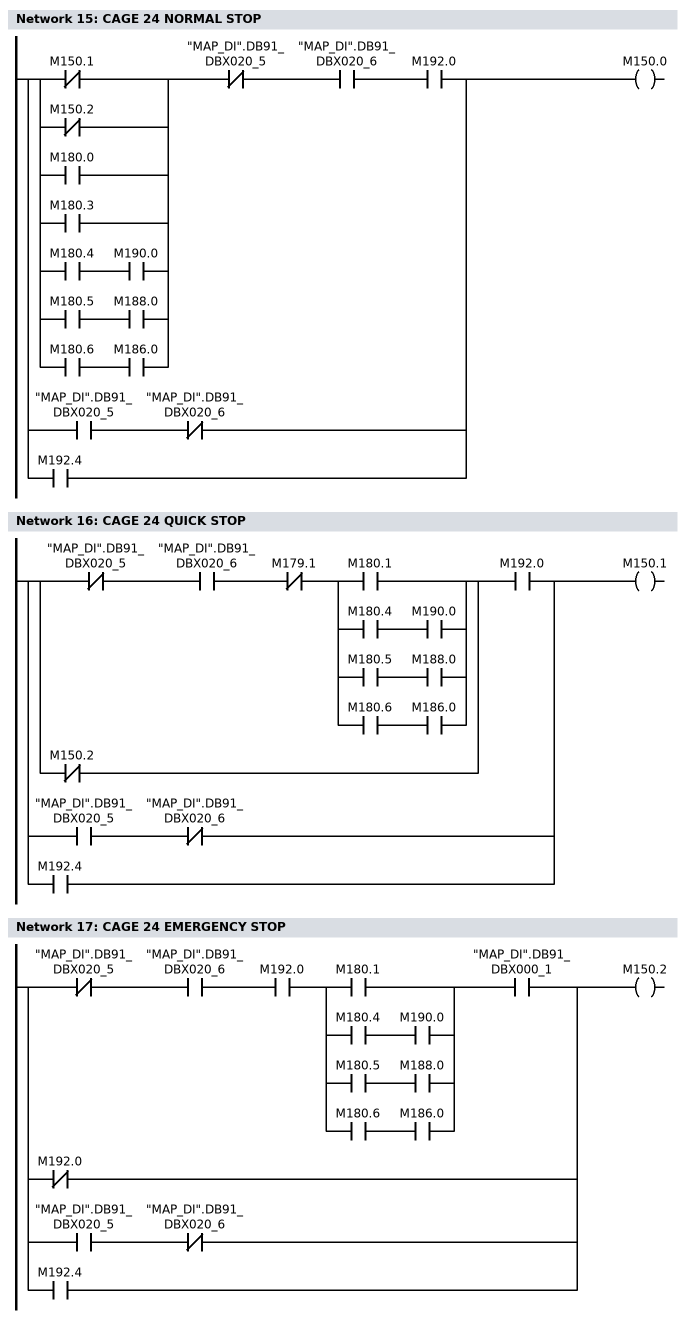
NETWORK
TITLE = CAGE 24 NORMAL STOP
      A(;
      ON    "M150.1";
      ON    "M150.2";
      O     "M180.0";
      O     "M180.3";
      O;
      A     "M180.4";
      A     "M190.0";
      O;
      A     "M180.5";
      A     "M188.0";
      O;
      A     "M180.6";
      A     "M186.0";
      );
      AN    "MAP_DI".DB91_DBX020_5;
      A     "MAP_DI".DB91_DBX020_6;
      A     "M192.0";
      O;
      A     "MAP_DI".DB91_DBX020_5;
      AN    "MAP_DI".DB91_DBX020_6;
      O     "M192.4";
      =     "M150.0";
NETWORK
TITLE = CAGE 24 QUICK STOP
      A(;
      AN    "MAP_DI".DB91_DBX020_5;
      A     "MAP_DI".DB91_DBX020_6;
      AN    "M179.1";
      A(;
      O     "M180.1";
      O;
      A     "M180.4";
      A     "M190.0";
      O;
      A     "M180.5";
      A     "M188.0";
      O;
      A     "M180.6";
      A     "M186.0";
      );
      ON    "M150.2";
      );
      A     "M192.0";
      O;
      A     "MAP_DI".DB91_DBX020_5;
      AN    "MAP_DI".DB91_DBX020_6;
      O     "M192.4";
      =     "M150.1";
NETWORK
TITLE = CAGE 24 EMERGENCY STOP
      AN    "MAP_DI".DB91_DBX020_5;
      A     "MAP_DI".DB91_DBX020_6;
      A     "M192.0";
      A(;
      O     "M180.1";
      O;
      A     "M180.4";
      A     "M190.0";
      O;
      A     "M180.5";
      A     "M188.0";
      O;
      A     "M180.6";
      A     "M186.0";
      );
      A     "MAP_DI".DB91_DBX000_1;
      ON    "M192.0";
      O;
      A     "MAP_DI".DB91_DBX020_5;
      AN    "MAP_DI".DB91_DBX020_6;
      O     "M192.4";
      =     "M150.2";
NETWORK
TITLE = CAGE 24 BRAKE PROPORTIONAL VALVE REFERENCE
      A     "M150.0";
      JC    _004;
      L     "Cage 24".DB15_DBD64;
      L     1.000000e+02;
      /R;
      L     2.764800e+04;
      *R;
      RND;
      JU    BRK;
_004: A     "M150.1";
      JC    _005;
      L     "Cage 24".DB15_DBD68;
      L     1.000000e+02;
      /R;
      L     2.764800e+04;
      *R;
      RND;
      JU    BRK;
_005: A     "M150.2";
      JC    _006;
      L     "Cage 24".DB15_DBD72;
      L     1.000000e+02;
      /R;
      L     2.764800e+04;
      *R;
      RND;
      JU    BRK;
_006: L     0;
BRK:  T     #Brake_value;
NETWORK
TITLE = SET POINT IN AMPER CALCULATION
      L     "Cage 24".DB15_DBD276;
      L     1.980000e+02;
      *R;
      L     1.000000e+02;
      /R;
      T     "Cage 24".DB15_DBD260;
NETWORK
TITLE = CURRENT CALCULATION
// (network holds code this reader does not know; not shown)
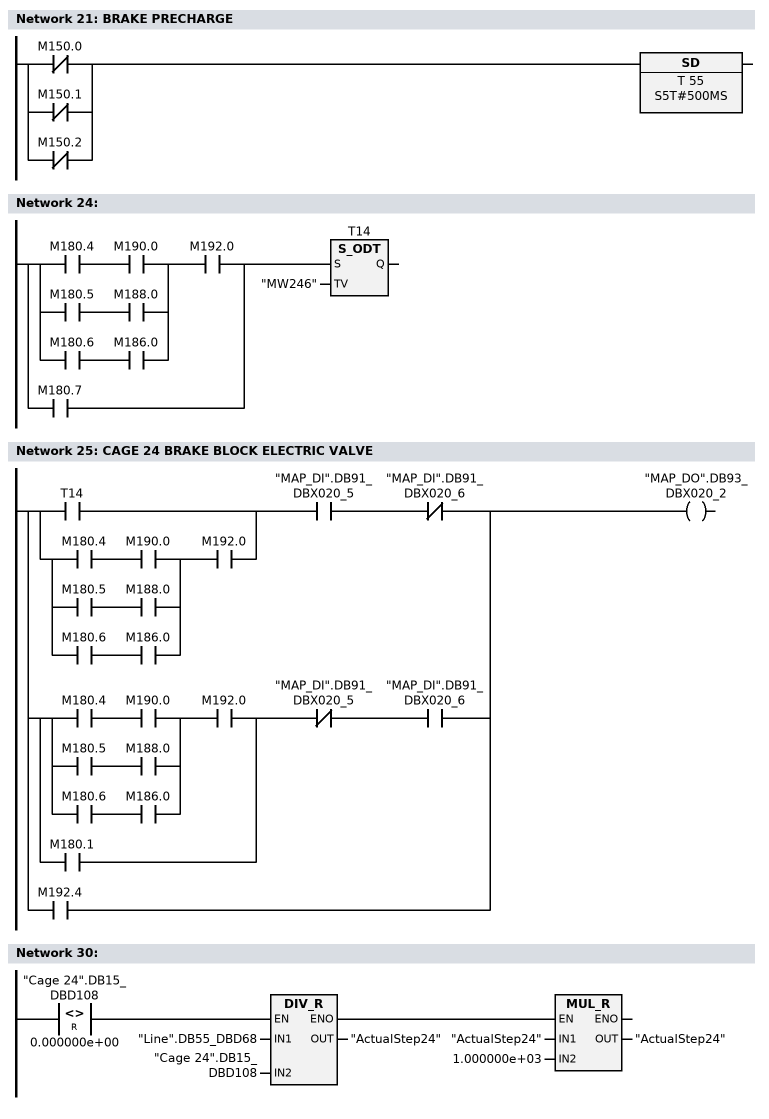
NETWORK
TITLE = BRAKE PRECHARGE
      ON    "M150.0";
      ON    "M150.1";
      ON    "M150.2";
      L     S5T#500MS;
      SD    T 55;
NETWORK
TITLE = BRAKE MODULATION CONTROL
      L     "Cage 24".DB15_DBD260;
      L     "Cage 24".DB15_DBD200;
      -R;
      T     "Cage 24".DB15_DBD264;
      L     "Cage 24".DB15_DBD268;
      *R;
      T     "Cage 24".DB15_DBD272;
      L     2.768400e+04;
      >R;
      JCN   _20d;
      L     2.768400e+04;
      T     "Cage 24".DB15_DBD272;
_20d: A     T 55;
      A     "M180.1";
      JCN   _20b;
      A(;
      L     "Cage 24".DB15_DBD272;
      L     0.000000e+00;
      <R;
      );
      JCN   _20a;
      L     0.000000e+00;
      T     "Cage 24".DB15_DBD272;
_20a: L     "Cage 24".DB15_DBD272;
      RND;
      JU    _20c;
_20b: L     #Brake_value;
_20c: T     "-659Y1";
NETWORK
TITLE = CAGE 24 BRAKE BLOCK OPEN ON-DELAY TIMER
      L     "Cage 24".DB15_DBD148;
      RND;
      ITB;
      L     W#16#2000;
      OW;
      T     "MW246";
NETWORK
TITLE =
      A(;
      A(;
      A     "M180.4";
      A     "M190.0";
      O;
      A     "M180.5";
      A     "M188.0";
      O;
      A     "M180.6";
      A     "M186.0";
      );
      A     "M192.0";
      O     "M180.7";
      );
      L     "MW246";
      SD    "T14";
      NOP   0;
      NOP   0;
      NOP   0;
      NOP   0;
NETWORK
TITLE = CAGE 24 BRAKE BLOCK ELECTRIC VALVE
      A(;
      O     "T14";
      O;
      A(;
      A     "M180.4";
      A     "M190.0";
      O;
      A     "M180.5";
      A     "M188.0";
      O;
      A     "M180.6";
      A     "M186.0";
      );
      A     "M192.0";
      );
      A     "MAP_DI".DB91_DBX020_5;
      AN    "MAP_DI".DB91_DBX020_6;
      O;
      A(;
      A(;
      A     "M180.4";
      A     "M190.0";
      O;
      A     "M180.5";
      A     "M188.0";
      O;
      A     "M180.6";
      A     "M186.0";
      );
      A     "M192.0";
      O     "M180.1";
      );
      AN    "MAP_DI".DB91_DBX020_5;
      A     "MAP_DI".DB91_DBX020_6;
      O     "M192.4";
      =     "MAP_DO".DB93_DBX020_2;
NETWORK
TITLE = CAGE 24 RPM TO HMI
      L     "Drives --> Plc".DB1_DBW1661;
      ITD;
      DTR;
      L     1.638400e+04;
      /R;
      L     2.400000e+02;
      *R;
      ABS;
      T     "Cage 24".DB15_DBD108;
NETWORK
TITLE = CAGE 24 MOTOR RPM TO HMI
      L     "Drives --> Plc".DB1_DBW1661;
      ITD;
      DTR;
      L     1.638400e+04;
      /R;
      L     1.460000e+03;
      *R;
      T     "Cage 24".DB15_DBD188;
NETWORK
TITLE = CAGE 24 MOTOR CURRENT TO HMI
      L     "Drives --> Plc".DB1_DBW1681;
      ITD;
      DTR;
      L     1.638400e+04;
      /R;
      L     1.980000e+02;
      *R;
      T     "Cage 24".DB15_DBD192;
NETWORK
TITLE = CAGE 24 MOTOR VOLTAGE TO HMI
      L     "Drives --> Plc".DB1_DBW1701;
      ITD;
      DTR;
      L     1.638400e+04;
      /R;
      L     4.000000e+02;
      *R;
      T     "Cage 24".DB15_DBD196;
NETWORK
TITLE =
      A(;
      A(;
      L     "Cage 24".DB15_DBD108;
      L     0.000000e+00;
      <>R;
      );
      JNB   _007;
      L     "Line".DB55_DBD68;
      L     "Cage 24".DB15_DBD108;
      /R;
      T     "ActualStep24";
      AN    OV;
      SAVE;
      CLR;
_007: A     BR;
      );
      JNB   _008;
      L     "ActualStep24";
      L     1.000000e+03;
      *R;
      T     "ActualStep24";
_008: NOP   0;
END_FUNCTION

FUNCTION "Cage 24 loading fase" : VOID	// FC 16
TITLE = CAGE 24 LOADING FASE FUNCTION
AUTHOR : Milesi
VERSION : 0.1
BEGIN
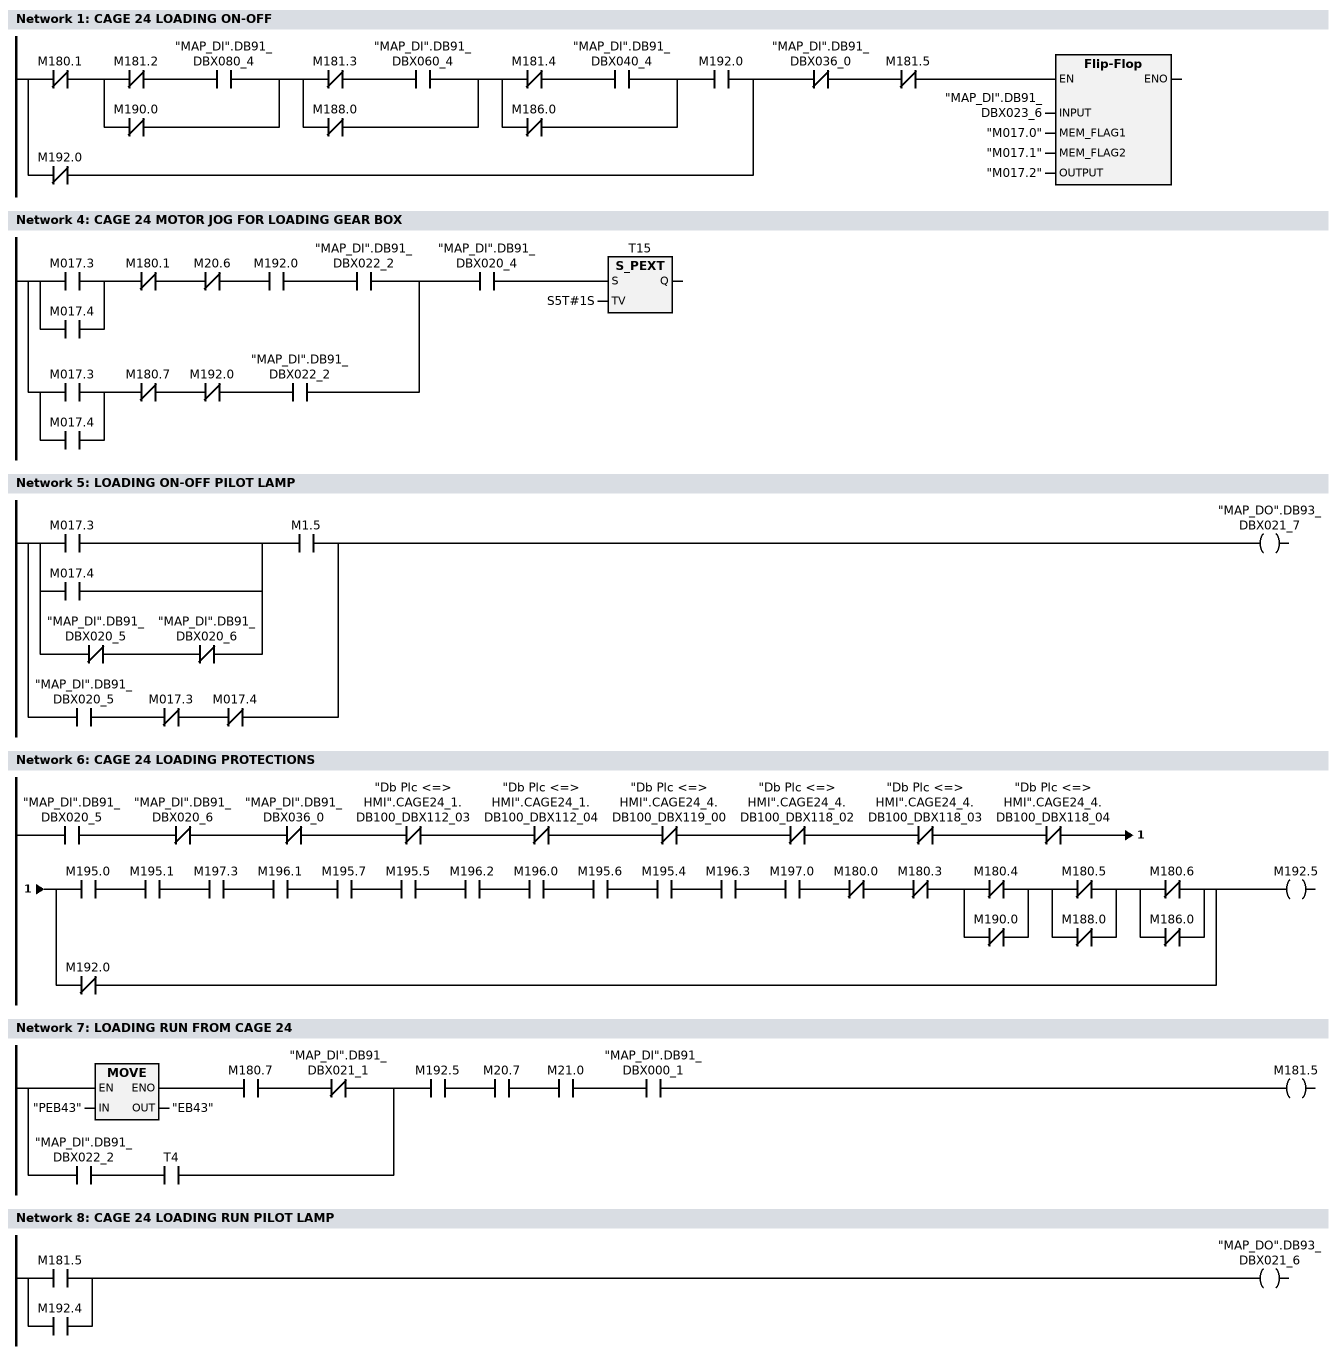
NETWORK
TITLE = CAGE 24 LOADING ON-OFF
      A(;
      AN    "M180.1";
      A(;
      AN    "M181.2";
      A     "MAP_DI".DB91_DBX080_4;
      ON    "M190.0";
      );
      A(;
      AN    "M181.3";
      A     "MAP_DI".DB91_DBX060_4;
      ON    "M188.0";
      );
      A(;
      AN    "M181.4";
      A     "MAP_DI".DB91_DBX040_4;
      ON    "M186.0";
      );
      A     "M192.0";
      ON    "M192.0";
      );
      AN    "MAP_DI".DB91_DBX036_0;
      AN    "M181.5";
      JNB   _001;
      CALL  "Flip-Flop" (
           INPUT                    := "MAP_DI".DB91_DBX023_6,
           MEM_FLAG1                := "M017.0",
           MEM_FLAG2                := "M017.1",
           OUTPUT                   := "M017.2");
_001: NOP   0;
NETWORK
TITLE = CAGE 24 LOADING ON
      A(;
      A(;
      A     "M017.2";
      AN    "M180.1";
      AN    "M20.6";
      A     "M192.0";
      O;
      AN    "M180.7";
      AN    "M192.0";
      );
      S     "MAP_DO".DB93_DBX020_0;
      A(;
      O     "MAP_DI".DB91_DBX020_5;
      O     "MAP_DO".DB93_DBX020_1;
      ON    "M017.2";
      );
      R     "MAP_DO".DB93_DBX020_0;
      A     "MAP_DO".DB93_DBX020_0;
      );
      S     "M017.3";
      A(;
      O     "MAP_DI".DB91_DBX020_5;
      ON    "M017.2";
      );
      R     "M017.3";
      NOP   0;
NETWORK
TITLE = CAGE 24 LOADING OFF
      A(;
      A(;
      AN    "M017.2";
      AN    "M20.6";
      A     "M192.0";
      O;
      AN    "M180.7";
      AN    "M192.0";
      );
      S     "MAP_DO".DB93_DBX020_1;
      A(;
      O     "MAP_DI".DB91_DBX020_6;
      O     "MAP_DO".DB93_DBX020_0;
      O     "M017.2";
      );
      R     "MAP_DO".DB93_DBX020_1;
      A     "MAP_DO".DB93_DBX020_1;
      );
      S     "M017.4";
      A(;
      O     "MAP_DI".DB91_DBX020_6;
      O     "M017.2";
      );
      R     "M017.4";
      NOP   0;
NETWORK
TITLE = CAGE 24 MOTOR JOG FOR LOADING GEAR BOX
      A(;
      A(;
      O     "M017.3";
      O     "M017.4";
      );
      AN    "M180.1";
      AN    "M20.6";
      A     "M192.0";
      A     "MAP_DI".DB91_DBX022_2;
      O;
      A(;
      O     "M017.3";
      O     "M017.4";
      );
      AN    "M180.7";
      AN    "M192.0";
      A     "MAP_DI".DB91_DBX022_2;
      );
      A     "MAP_DI".DB91_DBX020_4;
      L     S5T#1S;
      SE    "T15";
      NOP   0;
      NOP   0;
      NOP   0;
      NOP   0;
NETWORK
TITLE = LOADING ON-OFF PILOT LAMP
      A(;
      O     "M017.3";
      O     "M017.4";
      O;
      AN    "MAP_DI".DB91_DBX020_5;
      AN    "MAP_DI".DB91_DBX020_6;
      );
      A     "M1.5";
      O;
      A     "MAP_DI".DB91_DBX020_5;
      AN    "M017.3";
      AN    "M017.4";
      =     "MAP_DO".DB93_DBX021_7;
NETWORK
TITLE = CAGE 24 LOADING PROTECTIONS
      A     "MAP_DI".DB91_DBX020_5;
      AN    "MAP_DI".DB91_DBX020_6;
      AN    "MAP_DI".DB91_DBX036_0;
      AN    "Db Plc <=> HMI".CAGE24_1.DB100_DBX112_03;
      AN    "Db Plc <=> HMI".CAGE24_1.DB100_DBX112_04;
      AN    "Db Plc <=> HMI".CAGE24_4.DB100_DBX119_00;
      AN    "Db Plc <=> HMI".CAGE24_4.DB100_DBX118_02;
      AN    "Db Plc <=> HMI".CAGE24_4.DB100_DBX118_03;
      AN    "Db Plc <=> HMI".CAGE24_4.DB100_DBX118_04;
      A(;
      A     "M195.0";
      A     "M195.1";
      A     "M197.3";
      A     "M196.1";
      A     "M195.7";
      A     "M195.5";
      A     "M196.2";
      A     "M196.0";
      A     "M195.6";
      A     "M195.4";
      A     "M196.3";
      A     "M197.0";
      AN    "M180.0";
      AN    "M180.3";
      A(;
      ON    "M180.4";
      ON    "M190.0";
      );
      A(;
      ON    "M180.5";
      ON    "M188.0";
      );
      A(;
      ON    "M180.6";
      ON    "M186.0";
      );
      ON    "M192.0";
      );
      =     "M192.5";
NETWORK
TITLE = LOADING RUN FROM CAGE 24
      A(;
      A(;
      L     "PEB43";
      T     "EB43";
      SET;
      SAVE;
      CLR;
      A     BR;
      );
      A     "M180.7";
      AN    "MAP_DI".DB91_DBX021_1;
      O;
      A     "MAP_DI".DB91_DBX022_2;
      A     "T4";
      );
      A     "M192.5";
      A     "M20.7";
      A     "M21.0";
      A     "MAP_DI".DB91_DBX000_1;
      =     "M181.5";
NETWORK
TITLE = CAGE 24 LOADING RUN PILOT LAMP
      O     "M181.5";
      O     "M192.4";
      =     "MAP_DO".DB93_DBX021_6;
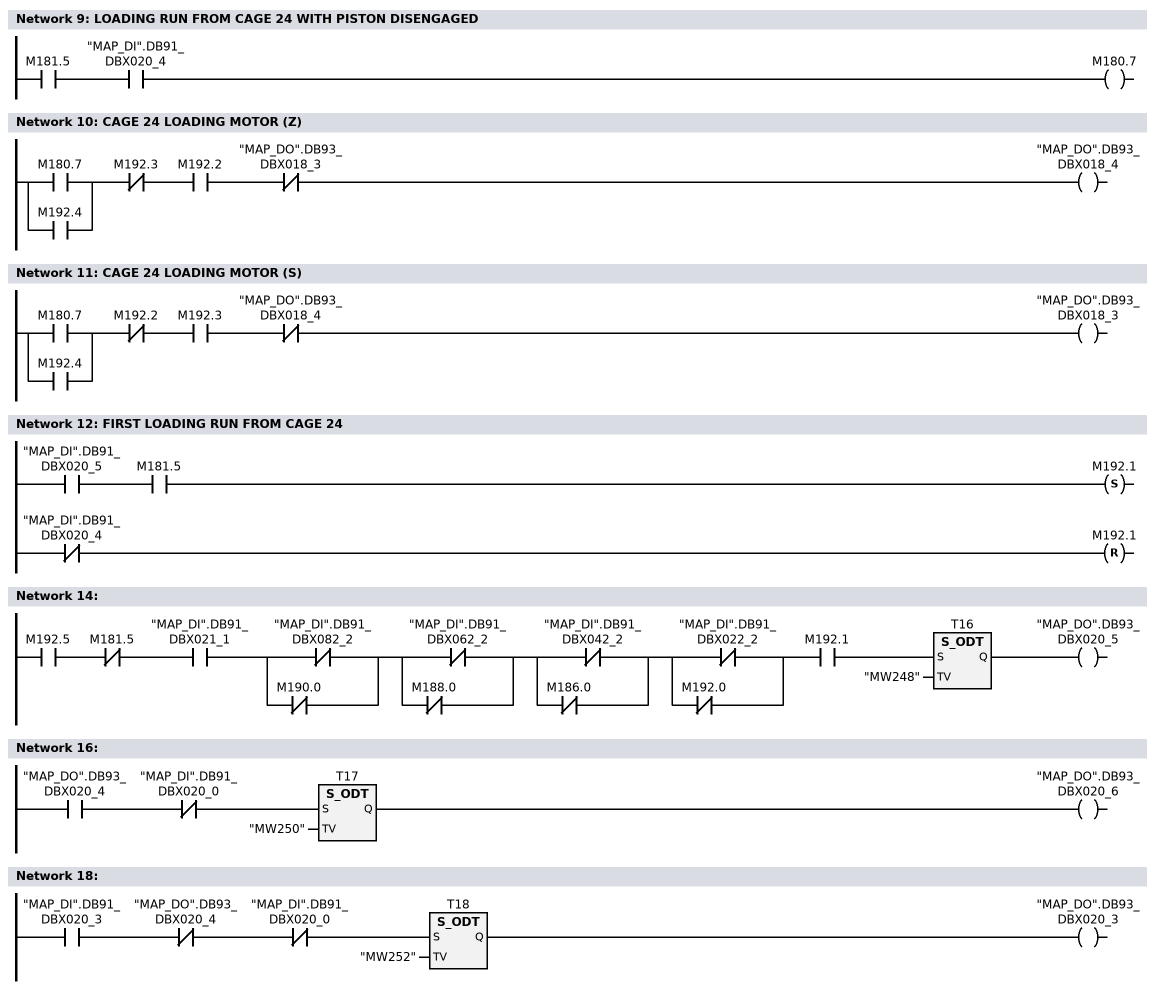
NETWORK
TITLE = LOADING RUN FROM CAGE 24 WITH PISTON DISENGAGED
      A     "M181.5";
      A     "MAP_DI".DB91_DBX020_4;
      =     "M180.7";
NETWORK
TITLE = CAGE 24 LOADING MOTOR (Z)
      A(;
      O     "M180.7";
      O     "M192.4";
      );
      AN    "M192.3";
      A     "M192.2";
      AN    "MAP_DO".DB93_DBX018_3;
      =     "MAP_DO".DB93_DBX018_4;
NETWORK
TITLE = CAGE 24 LOADING MOTOR (S)
      A(;
      O     "M180.7";
      O     "M192.4";
      );
      AN    "M192.2";
      A     "M192.3";
      AN    "MAP_DO".DB93_DBX018_4;
      =     "MAP_DO".DB93_DBX018_3;
NETWORK
TITLE = FIRST LOADING RUN FROM CAGE 24
      A     "MAP_DI".DB91_DBX020_5;
      A     "M181.5";
      S     "M192.1";
      AN    "MAP_DI".DB91_DBX020_4;
      R     "M192.1";
      NOP   0;
NETWORK
TITLE = CAGE 24 PISTON ENGAGING INTO CAGE
      L     "Cage 24".DB15_DBD152;
      RND;
      ITB;
      L     W#16#2000;
      OW;
      T     "MW248";
NETWORK
TITLE =
      A     "M192.5";
      AN    "M181.5";
      A     "MAP_DI".DB91_DBX021_1;
      A(;
      ON    "MAP_DI".DB91_DBX082_2;
      ON    "M190.0";
      );
      A(;
      ON    "MAP_DI".DB91_DBX062_2;
      ON    "M188.0";
      );
      A(;
      ON    "MAP_DI".DB91_DBX042_2;
      ON    "M186.0";
      );
      A(;
      ON    "MAP_DI".DB91_DBX022_2;
      ON    "M192.0";
      );
      A     "M192.1";
      L     "MW248";
      SD    "T16";
      NOP   0;
      NOP   0;
      NOP   0;
      A     "T16";
      =     "MAP_DO".DB93_DBX020_5;
NETWORK
TITLE = CAGE 24 PISTON DISENGAGING FROM CAGE
      L     "Cage 24".DB15_DBD144;
      RND;
      ITB;
      L     W#16#2000;
      OW;
      T     "MW250";
NETWORK
TITLE =
      A     "MAP_DO".DB93_DBX020_4;
      AN    "MAP_DI".DB91_DBX020_0;
      L     "MW250";
      SD    "T17";
      NOP   0;
      NOP   0;
      NOP   0;
      A     "T17";
      =     "MAP_DO".DB93_DBX020_6;
NETWORK
TITLE = CAGE 24 AIR INLET INTO CAGE
      L     "Cage 24".DB15_DBD156;
      RND;
      ITB;
      L     W#16#2000;
      OW;
      T     "MW252";
NETWORK
TITLE =
      A     "MAP_DI".DB91_DBX020_3;
      AN    "MAP_DO".DB93_DBX020_4;
      AN    "MAP_DI".DB91_DBX020_0;
      L     "MW252";
      SD    "T18";
      NOP   0;
      NOP   0;
      NOP   0;
      A     "T18";
      =     "MAP_DO".DB93_DBX020_3;
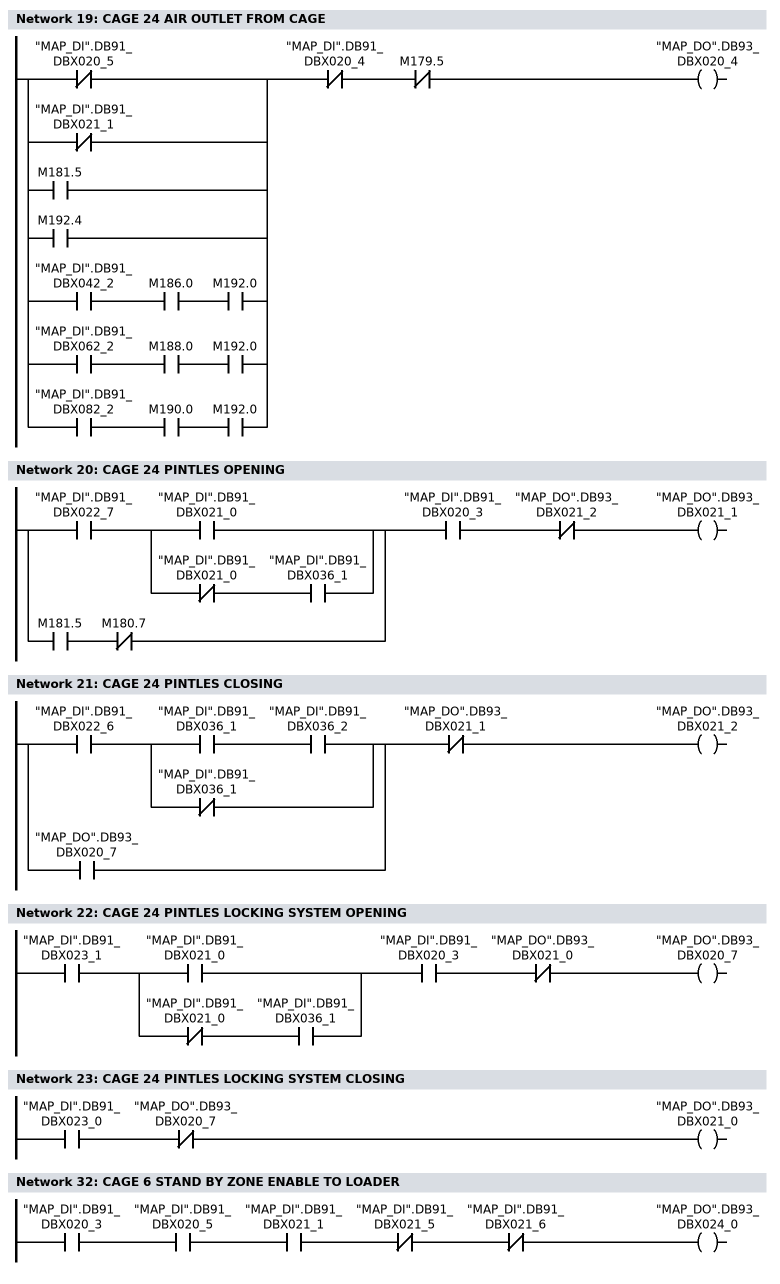
NETWORK
TITLE = CAGE 24 AIR OUTLET FROM CAGE
      A(;
      ON    "MAP_DI".DB91_DBX020_5;
      ON    "MAP_DI".DB91_DBX021_1;
      O     "M181.5";
      O     "M192.4";
      O;
      A     "MAP_DI".DB91_DBX042_2;
      A     "M186.0";
      A     "M192.0";
      O;
      A     "MAP_DI".DB91_DBX062_2;
      A     "M188.0";
      A     "M192.0";
      O;
      A     "MAP_DI".DB91_DBX082_2;
      A     "M190.0";
      A     "M192.0";
      );
      AN    "MAP_DI".DB91_DBX020_4;
      AN    "M179.5";
      =     "MAP_DO".DB93_DBX020_4;
NETWORK
TITLE = CAGE 24 PINTLES OPENING
      A(;
      A     "MAP_DI".DB91_DBX022_7;
      A(;
      O     "MAP_DI".DB91_DBX021_0;
      O;
      AN    "MAP_DI".DB91_DBX021_0;
      A     "MAP_DI".DB91_DBX036_1;
      );
      O;
      A     "M181.5";
      AN    "M180.7";
      );
      A     "MAP_DI".DB91_DBX020_3;
      AN    "MAP_DO".DB93_DBX021_2;
      =     "MAP_DO".DB93_DBX021_1;
NETWORK
TITLE = CAGE 24 PINTLES CLOSING
      A(;
      A     "MAP_DI".DB91_DBX022_6;
      A(;
      A     "MAP_DI".DB91_DBX036_1;
      A     "MAP_DI".DB91_DBX036_2;
      ON    "MAP_DI".DB91_DBX036_1;
      );
      O     "MAP_DO".DB93_DBX020_7;
      );
      AN    "MAP_DO".DB93_DBX021_1;
      =     "MAP_DO".DB93_DBX021_2;
NETWORK
TITLE = CAGE 24 PINTLES LOCKING SYSTEM OPENING
      A     "MAP_DI".DB91_DBX023_1;
      A(;
      O     "MAP_DI".DB91_DBX021_0;
      O;
      AN    "MAP_DI".DB91_DBX021_0;
      A     "MAP_DI".DB91_DBX036_1;
      );
      A     "MAP_DI".DB91_DBX020_3;
      AN    "MAP_DO".DB93_DBX021_0;
      =     "MAP_DO".DB93_DBX020_7;
NETWORK
TITLE = CAGE 24 PINTLES LOCKING SYSTEM CLOSING
      A     "MAP_DI".DB91_DBX023_0;
      AN    "MAP_DO".DB93_DBX020_7;
      =     "MAP_DO".DB93_DBX021_0;
NETWORK
TITLE = CAGE 24 PLATFORM UP
NETWORK
TITLE = CAGE 24 PLATFORM DOWN
NETWORK
TITLE = CAGE 24 EVEN BOBBINS ROTATION FOR LOADING MACHINE
NETWORK
TITLE = CAGE 24 EVEN BOBBINS ROTATION FOR LOADING PLATFORM
NETWORK
TITLE = CAGE 24 ODD BOBBINS ROTATION FOR LOADING MACHINE
NETWORK
TITLE = CAGE 24 ODD BOBBINS ROTATION FOR LOADING PLATFORM
NETWORK
TITLE = CAGE 24 BOBBIN ROTATION FOR LOADING MACHINE PILOT LAMP
NETWORK
TITLE = CAGE 24 LOADING PUMP
NETWORK
TITLE = CAGE 6 STAND BY ZONE ENABLE TO LOADER
      A     "MAP_DI".DB91_DBX020_3;
      A     "MAP_DI".DB91_DBX020_5;
      A     "MAP_DI".DB91_DBX021_1;
      AN    "MAP_DI".DB91_DBX021_5;
      AN    "MAP_DI".DB91_DBX021_6;
      =     "MAP_DO".DB93_DBX024_0;
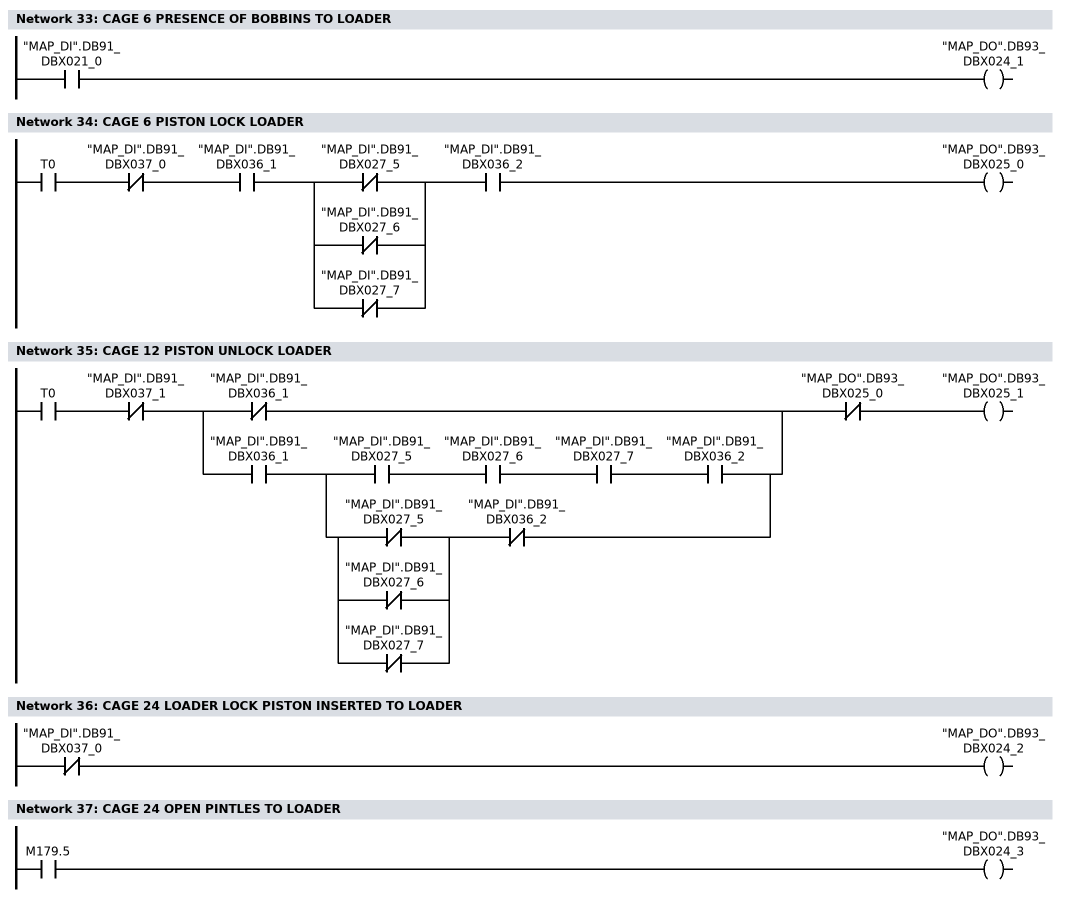
NETWORK
TITLE = CAGE 6 PRESENCE OF BOBBINS TO LOADER
      A     "MAP_DI".DB91_DBX021_0;
      =     "MAP_DO".DB93_DBX024_1;
NETWORK
TITLE = CAGE 6 PISTON LOCK LOADER
      A     "T0";
      AN    "MAP_DI".DB91_DBX037_0;
      A     "MAP_DI".DB91_DBX036_1;
      A(;
      ON    "MAP_DI".DB91_DBX027_5;
      ON    "MAP_DI".DB91_DBX027_6;
      ON    "MAP_DI".DB91_DBX027_7;
      );
      A     "MAP_DI".DB91_DBX036_2;
      =     "MAP_DO".DB93_DBX025_0;
NETWORK
TITLE = CAGE 12 PISTON UNLOCK LOADER
      A     "T0";
      AN    "MAP_DI".DB91_DBX037_1;
      A(;
      ON    "MAP_DI".DB91_DBX036_1;
      O;
      A     "MAP_DI".DB91_DBX036_1;
      A(;
      A     "MAP_DI".DB91_DBX027_5;
      A     "MAP_DI".DB91_DBX027_6;
      A     "MAP_DI".DB91_DBX027_7;
      A     "MAP_DI".DB91_DBX036_2;
      O;
      A(;
      ON    "MAP_DI".DB91_DBX027_5;
      ON    "MAP_DI".DB91_DBX027_6;
      ON    "MAP_DI".DB91_DBX027_7;
      );
      AN    "MAP_DI".DB91_DBX036_2;
      );
      );
      AN    "MAP_DO".DB93_DBX025_0;
      =     "MAP_DO".DB93_DBX025_1;
NETWORK
TITLE = CAGE 24 LOADER LOCK PISTON INSERTED TO LOADER 
      AN    "MAP_DI".DB91_DBX037_0;
      =     "MAP_DO".DB93_DBX024_2;
NETWORK
TITLE = CAGE 24 OPEN PINTLES TO LOADER
      A     "M179.5";
      =     "MAP_DO".DB93_DBX024_3;
END_FUNCTION

FUNCTION "Cage 24 preforming alarm" : VOID	// FC 17
TITLE = CAGE 24 PREFORMING ALARMS FUNCTION
AUTHOR : Milesi
VERSION : 0.1
BEGIN
NETWORK
TITLE = CAGE 24 PREFORMING MOTOR DRIVE PROFIBUS SLAVE 6 FAULT
      A(;
      L     "MB304";
      L     6;
      ==I;
      );
      AN    "M300.5";
      S     "Db Plc <=> HMI".PROFIBUS.DB100_DBX101_5;
NETWORK
TITLE = CAGE 24 PREFORMING MOTOR BRAKE OVERLOAD
      A     "T0";
      A     "MAP_DI".DB91_DBX018_4;
      A     "M193.3";
      =     "Db Plc <=> HMI".CAGE24_4.DB100_DBX119_04;
NETWORK
TITLE = CAGE 24 PREFORMING MOTOR BLOWER OVERLOAD
      A     "T0";
      A     "MAP_DI".DB91_DBX018_5;
      A     "M193.3";
      =     "Db Plc <=> HMI".CAGE24_4.DB100_DBX119_05;
NETWORK
TITLE = CAGE 24 PREFORMING OPEN GUARD
      A     "T0";
      A     "M180.1";
      AN    "MAP_DI".DB91_DBX024_6;
      A     "M193.3";
      S     "M174.3";
NETWORK
TITLE =
      A     "T0";
      A(;
      ON    "MAP_DI".DB91_DBX024_6;
      O     "M174.3";
      );
      A     "M193.3";
      =     "Db Plc <=> HMI".CAGE24_4.DB100_DBX119_06;
NETWORK
TITLE = CAGE 24 PREFORMING MOTOR DRIVE FAULT
      A     "T0";
      A     "Drives --> Plc".CAGE_24_PREF_STATUS_W1.DB1_DBX121_3;
      A     "M193.3";
      S     "Db Plc <=> HMI".CAGE24_4.DB100_DBX119_07;
NETWORK
TITLE = CAGE 24 PREFORMING GENERAL ALARM
      AN    "Db Plc <=> HMI".PROFIBUS.DB100_DBX101_5;
      AN    "Db Plc <=> HMI".CAGE24_4.DB100_DBX119_04;
      AN    "Db Plc <=> HMI".CAGE24_4.DB100_DBX119_05;
      AN    "Db Plc <=> HMI".CAGE24_4.DB100_DBX119_06;
      AN    "Db Plc <=> HMI".CAGE24_4.DB100_DBX119_07;
      =     "M195.4";
END_FUNCTION

FUNCTION "Cage 24 preforming unit" : VOID	// FC 18
TITLE = CAGE 24 PREFORMING UNIT FUNCTION
AUTHOR : Milesi
VERSION : 0.1
BEGIN
NETWORK
TITLE = CAGE 24 PREFORMING OFF
      A(;
      L     "Cage 24 preforming".DB18_DBW2;
      L     0;
      ==I;
      );
      AN    "M180.1";
      JNB   _001;
      R     "M193.3";
      R     "M193.4";
      R     "M193.5";
_001: NOP   0;
NETWORK
TITLE = CAGE 24 PREFORMING Z ROTATION
      A(;
      L     "Cage 24 preforming".DB18_DBW2;
      L     1;
      ==I;
      );
      AN    "M180.1";
      JNB   _002;
      S     "M193.3";
      S     "M193.4";
      R     "M193.5";
_002: NOP   0;
NETWORK
TITLE = CAGE 24 PREFORMING S ROTATION
      A(;
      L     "Cage 24 preforming".DB18_DBW2;
      L     2;
      ==I;
      );
      AN    "M180.1";
      JNB   _003;
      S     "M193.3";
      S     "M193.5";
      R     "M193.4";
_003: NOP   0;
NETWORK
TITLE = CAGE 24 PREFORMING MOTOR DRIVE RUN
      A(;
      O     "M180.1";
      O     "M21.3";
      );
      AN    "Db Plc <=> HMI".CAGE24_4.DB100_DBX119_07;
      A     "M193.3";
      =     "Plc --> Drives".CAGE_24_PREF_CONTROL_W1.DB2_DBX121_0;
      =     "Plc --> Drives".CAGE_24_PREF_CONTROL_W1.DB2_DBX121_3;
NETWORK
TITLE = CAGE 24 PREFORMING MOTOR BLOWER
      A     "Plc --> Drives".CAGE_24_PREF_CONTROL_W1.DB2_DBX121_0;
      AN    "Db Plc <=> HMI".CAGE24_4.DB100_DBX119_05;
      =     "MAP_DO".DB93_DBX018_1;
NETWORK
TITLE = CAGE 24 PREFORMING MOTOR ELECTRIC BRAKE RELAY
      A(;
      O     "Plc --> Drives".CAGE_24_PREF_CONTROL_W1.DB2_DBX121_0;
      O     "MAP_DI".DB91_DBX024_7;
      );
      AN    "Db Plc <=> HMI".CAGE24_4.DB100_DBX119_05;
      =     "MAP_DO".DB93_DBX018_0;
NETWORK
TITLE = CAGE 24 PREFORMING MOTOR REFERENCE
//Max Linear Speed = 40 m/min
//Max Die Rpm = 147.68
//
//Max Linear Speed             40000
//---------------- = Die Lay = ------ = 270.85
//  Max Die Rpm                147.68
//
//                               Max Linear Speed
//Max Die Rpm = 147.68 = 16384 = ---------------- * K
//                                   Die Lay
//
//    Die Lay * 16384   270.85 * 16384
//K = ---------------- = ------------- = 110940.16
//    Max Linear Speed        40
// (network holds code this reader does not know; not shown)
NETWORK
TITLE = CAGE 24 PREFORMING RPM TO HMI
      L     "Drives --> Plc".DB1_DBW126;
      ITD;
      DTR;
      L     1.638400e+04;
      /R;
      L     1.476800e+02;
      *R;
      ABS;
      T     "Cage 24 preforming".DB18_DBD108;
NETWORK
TITLE = CAGE 24 PREFORMING MOTOR RPM TO HMI
      L     "Drives --> Plc".DB1_DBW126;
      ITD;
      DTR;
      L     1.638400e+04;
      /R;
      L     1.420000e+03;
      *R;
      T     "Cage 24 preforming".DB18_DBD188;
NETWORK
TITLE = CAGE 24 PREFORMING MOTOR CURRENT TO HMI
//TORQUE FEEDBACK = 150% = MOTOR CURRENT * 1.5
      L     "Drives --> Plc".DB1_DBW128;
      ITD;
      DTR;
      L     1.638400e+04;
      /R;
      L     3.400000e+00;
      *R;
      T     "Cage 24 preforming".DB18_DBD192;
NETWORK
TITLE = CAGE 24 PREFORMING MOTOR VOLTAGE TO HMI
      L     "Drives --> Plc".DB1_DBW130;
      ITD;
      DTR;
      L     1.638400e+04;
      /R;
      L     4.000000e+02;
      *R;
      T     "Cage 24 preforming".DB18_DBD196;
END_FUNCTION

FUNCTION "Cage 18 alarms" : VOID	// FC 19
TITLE = CAGE 18 ALARMS FUNCTION
AUTHOR : Milesi
VERSION : 0.1
VAR_TEMP
  T4_time : WORD ;
END_VAR
BEGIN
NETWORK
TITLE = CAGE 18 MOTOR DRIVE PROFIBUS SLAVE 9 FAULT
      A(;
      L     "MB304";
      L     9;
      ==I;
      );
      AN    "M300.5";
      S     "Db Plc <=> HMI".PROFIBUS.DB100_DBX100_0;
NETWORK
TITLE = CAGE 18 ET200M PROFIBUS SLAVE 22 FAULT
      A(;
      L     "MB304";
      L     22;
      ==I;
      );
      AN    "M300.5";
      S     "Db Plc <=> HMI".PROFIBUS.DB100_DBX100_6;
NETWORK
TITLE = CAGE 18 OPEN FRONT GUARD ALARM
      A     "T0";
      A     "M180.1";
      AN    "MAP_DI".DB91_DBX041_6;
      A     "M186.0";
      S     "M173.4";
NETWORK
TITLE =
      A     "T0";
      A(;
      ON    "MAP_DI".DB91_DBX041_6;
      O     "M173.4";
      );
      A     "M186.0";
      =     "Db Plc <=> HMI".CAGE18_1.DB100_DBX120_00;
NETWORK
TITLE = CAGE 18 PRESENCE OF MAN ALARM
      A     "T0";
      AN    "MAP_DI".DB91_DBX041_7;
      AN    "M180.1";
      A     "M186.0";
      =     "Db Plc <=> HMI".CAGE18_1.DB100_DBX120_01;
NETWORK
TITLE = CAGE 18 LOADING ENGAGED
      A     "T0";
      A     "MAP_DI".DB91_DBX040_5;
      AN    "MAP_DI".DB91_DBX040_6;
      A     "M16.2";
      =     "Db Plc <=> HMI".CAGE18_1.DB100_DBX120_02;
NETWORK
TITLE = CAGE 18 LOADING GEAR BOX NOT ENGAGED
      A     "T0";
      AN    "MAP_DI".DB91_DBX040_5;
      AN    "MAP_DI".DB91_DBX040_6;
      =     "Db Plc <=> HMI".CAGE18_1.DB100_DBX120_03;
NETWORK
TITLE = CAGE 18 LOADING MOTOR OVERLOAD
      A     "T0";
      A     "MAP_DI".DB91_DBX038_2;
      =     "Db Plc <=> HMI".CAGE18_1.DB100_DBX120_04;
NETWORK
TITLE = CAGE 18 AIR PIPE NOT IN POSITION
      A     "T0";
      A     "M180.1";
      AN    "MAP_DI".DB91_DBX040_7;
      A     "M186.0";
      S     "M173.5";
NETWORK
TITLE =
      A     "T0";
      A(;
      ON    "MAP_DI".DB91_DBX040_7;
      O     "M173.5";
      );
      =     "Db Plc <=> HMI".CAGE18_1.DB100_DBX120_05;
NETWORK
TITLE = CAGE 18 PISTON INSIDE CAGE
      A     "T0";
      A     "M180.1";
      AN    "MAP_DI".DB91_DBX040_4;
      A     "M186.0";
      S     "M173.3";
NETWORK
TITLE =
      A     "T0";
      A(;
      ON    "MAP_DI".DB91_DBX040_4;
      O     "M173.3";
      );
      =     "Db Plc <=> HMI".CAGE18_1.DB100_DBX120_07;
NETWORK
TITLE = CAGE 18 24VDC POWER SUPPLY OVERLOAD
      A     "T0";
      AN    "MAP_DI".DB91_DBX038_1;
      =     "Db Plc <=> HMI".CAGE18_1.DB100_DBX121_00;
NETWORK
TITLE = CAGE 18 230VAC POWER SUPPLY OVERLOAD
      A     "T0";
      AN    "MAP_DI".DB91_DBX038_0;
      =     "Db Plc <=> HMI".CAGE18_1.DB100_DBX121_01;
NETWORK
TITLE = CAGE 18 MOTOR BLOWER OVERLOAD
      A     "T0";
      A     "MAP_DI".DB91_DBX038_3;
      =     "Db Plc <=> HMI".CAGE18_1.DB100_DBX121_02;
NETWORK
TITLE = CAGE 18 LOADING PLATFORM MOTOR OVERLOAD
NETWORK
TITLE = CAGE 18 GUARD BLOWER MOTOR OVERLOAD
      A     "T0";
      A     "MAP_DI".DB91_DBX038_7;
      =     "Db Plc <=> HMI".CAGE18_1.DB100_DBX121_05;
NETWORK
TITLE = CAGE 18 OPEN FRONT DOOR
//      U(    
//      U(    
//      U     T      0
//      U     M    178.0
//      O     M    180.1
//      O     M     21.3
//      )     
//      L     S5T#2S
//      SE    T     25
//      NOP   0
//      NOP   0
//      NOP   0
//      U     T     25
//      )     
//      UN    DB91.DBX   41.3
//      U     M    186.0
//      S     DB100.DBX  121.6
NETWORK
TITLE = CAGE 18 OPEN REAR DOORS
      A     "T0";
      A     "M180.1";
      AN    "MAP_DI".DB91_DBX041_4;
      A     "M186.0";
      S     "M173.6";
NETWORK
TITLE =
      A     "T0";
      A(;
      ON    "MAP_DI".DB91_DBX041_4;
      O     "M173.6";
      );
      A     "M186.0";
      =     "Db Plc <=> HMI".CAGE18_1.DB100_DBX121_07;
NETWORK
TITLE = CAGE 18 BREAK WIRE FROM RING 
      A     "T0";
      A     "T1";
      AN    "MAP_DI".DB91_DBX041_2;
      A     "M186.0";
      S     "Db Plc <=> HMI".CAGE18_3.DB100_DBX125_06;
NETWORK
TITLE = CAGE 18 MAIN AIR MINIMUM PRESSURE
      A     "T0";
      A     "M180.1";
      AN    "MAP_DI".DB91_DBX040_2;
      A     "M186.0";
      S     "M173.7";
NETWORK
TITLE =
      A     "T0";
      A(;
      ON    "MAP_DI".DB91_DBX040_2;
      O     "M173.7";
      );
      =     "Db Plc <=> HMI".CAGE18_4.DB100_DBX126_00;
NETWORK
TITLE = CAGE 18 BOBBIN BRAKES AIR TANK MINIMUM PRESSURE
      A     "T0";
      AN    "Db Plc <=> HMI".PROFIBUS.DB100_DBX100_6;
      AN    "MAP_DI".DB91_DBX047_0;
      A     "M186.0";
      S     "Db Plc <=> HMI".CAGE18_4.DB100_DBX126_01;
NETWORK
TITLE = CAGE 18 LINE 1 PINTLES OPEN
      A     "T0";
      A     "M180.1";
      AN    "MAP_DI".DB91_DBX047_1;
      A     "M186.0";
      S     "M174.0";
NETWORK
TITLE =
      A     "T0";
      A(;
      ON    "MAP_DI".DB91_DBX047_1;
      O     "M174.0";
      );
      =     "Db Plc <=> HMI".CAGE18_4.DB100_DBX126_02;
NETWORK
TITLE = CAGE 18 LINE 2 PINTLES OPEN
      A     "T0";
      A     "M180.1";
      AN    "MAP_DI".DB91_DBX047_2;
      A     "M186.0";
      S     "M174.1";
NETWORK
TITLE =
      A     "T0";
      A(;
      ON    "MAP_DI".DB91_DBX047_2;
      O     "M174.1";
      );
      =     "Db Plc <=> HMI".CAGE18_4.DB100_DBX126_03;
NETWORK
TITLE = CAGE 18 LINE 3 PINTLES OPEN
      A     "T0";
      A     "M180.1";
      AN    "MAP_DI".DB91_DBX047_3;
      A     "M186.0";
      S     "M174.2";
NETWORK
TITLE =
      A     "T0";
      A(;
      ON    "MAP_DI".DB91_DBX047_3;
      O     "M174.2";
      );
      =     "Db Plc <=> HMI".CAGE18_4.DB100_DBX126_04;
NETWORK
TITLE = CAGE 18 OPEN PINTLES LAMP
      ON    "MAP_DI".DB91_DBX047_1;
      ON    "MAP_DI".DB91_DBX047_2;
      ON    "MAP_DI".DB91_DBX047_3;
      =     "M179.4";
      =     "MAP_DO".DB93_DBX032_0;
NETWORK
TITLE = CAGE 18 MOTOR DRIVE FAULT
      A     "T0";
      A     "Drives --> Plc".CAGE_18_STATUS_W1.DB1_DBX241_3;
      S     "Db Plc <=> HMI".CAGE18_4.DB100_DBX126_05;
NETWORK
TITLE = CAGE 18 MOTOR OVERTEMPERATURE
      A     "T0";
      A     "Drives --> Plc".CAGE_18_STATUS_W2.DB1_DBX242_1;
      S     "Db Plc <=> HMI".CAGE18_4.DB100_DBX126_06;
NETWORK
TITLE = CAGE 18 OVERSPEED
      A     "T0";
      A     "M180.1";
      A(;
      L     "Cage 18".DB20_DBD108;
      L     2.850000e+02;
      >=R;
      );
      A     "M186.0";
      S     "Db Plc <=> HMI".CAGE18_4.DB100_DBX126_07;
NETWORK
TITLE = CAGE 18 BRAKES CONTROL
      A     "T0";
      A     "T2";
      AN    "MAP_DI".DB91_DBX040_1;
      A     "M186.0";
      S     "Db Plc <=> HMI".CAGE18_4.DB100_DBX127_00;
NETWORK
TITLE = CAGE 18 PLATFORM UP
NETWORK
TITLE = CAGE 18 HIDRAULIC UNIT MINIMUM OIL LEVEL  
NETWORK
TITLE = CAGE 18 GENERAL ALARM
      AN    "Db Plc <=> HMI".PROFIBUS.DB100_DBX100_0;
      AN    "Db Plc <=> HMI".PROFIBUS.DB100_DBX100_6;
      AN    "Db Plc <=> HMI".CAGE18_1.DB100_DBX120_00;
      AN    "Db Plc <=> HMI".CAGE18_1.DB100_DBX120_01;
      AN    "Db Plc <=> HMI".CAGE18_1.DB100_DBX120_03;
      AN    "Db Plc <=> HMI".CAGE18_1.DB100_DBX120_05;
      AN    "Db Plc <=> HMI".CAGE18_1.DB100_DBX120_07;
      AN    "Db Plc <=> HMI".CAGE18_1.DB100_DBX121_00;
      AN    "Db Plc <=> HMI".CAGE18_1.DB100_DBX121_01;
      AN    "Db Plc <=> HMI".CAGE18_1.DB100_DBX121_02;
      AN    "Db Plc <=> HMI".CAGE18_1.DB100_DBX121_06;
      AN    "Db Plc <=> HMI".CAGE18_1.DB100_DBX121_07;
      AN    "Db Plc <=> HMI".CAGE18_2.DB100_DBX122_00;
      AN    "Db Plc <=> HMI".CAGE18_2.DB100_DBX122_01;
      AN    "Db Plc <=> HMI".CAGE18_2.DB100_DBX122_02;
      AN    "Db Plc <=> HMI".CAGE18_2.DB100_DBX122_03;
      AN    "Db Plc <=> HMI".CAGE18_2.DB100_DBX122_04;
      AN    "Db Plc <=> HMI".CAGE18_2.DB100_DBX122_05;
      AN    "Db Plc <=> HMI".CAGE18_2.DB100_DBX122_06;
      AN    "Db Plc <=> HMI".CAGE18_2.DB100_DBX122_07;
      AN    "Db Plc <=> HMI".CAGE18_2.DB100_DBX123_00;
      AN    "Db Plc <=> HMI".CAGE18_2.DB100_DBX123_01;
      AN    "Db Plc <=> HMI".CAGE18_2.DB100_DBX123_02;
      AN    "Db Plc <=> HMI".CAGE18_2.DB100_DBX123_03;
      AN    "Db Plc <=> HMI".CAGE18_2.DB100_DBX123_04;
      AN    "Db Plc <=> HMI".CAGE18_2.DB100_DBX123_05;
      AN    "Db Plc <=> HMI".CAGE18_2.DB100_DBX123_06;
      AN    "Db Plc <=> HMI".CAGE18_2.DB100_DBX123_07;
      AN    "Db Plc <=> HMI".CAGE18_3.DB100_DBX124_00;
      AN    "Db Plc <=> HMI".CAGE18_3.DB100_DBX124_01;
      AN    "Db Plc <=> HMI".CAGE18_3.DB100_DBX125_06;
      AN    "Db Plc <=> HMI".CAGE18_3.DB100_DBX125_07;
      AN    "Db Plc <=> HMI".CAGE18_4.DB100_DBX126_00;
      AN    "Db Plc <=> HMI".CAGE18_4.DB100_DBX126_01;
      AN    "Db Plc <=> HMI".CAGE18_4.DB100_DBX126_02;
      AN    "Db Plc <=> HMI".CAGE18_4.DB100_DBX126_03;
      AN    "Db Plc <=> HMI".CAGE18_4.DB100_DBX126_04;
      AN    "Db Plc <=> HMI".CAGE18_4.DB100_DBX126_05;
      AN    "Db Plc <=> HMI".CAGE18_4.DB100_DBX126_06;
      AN    "Db Plc <=> HMI".CAGE18_4.DB100_DBX126_07;
      AN    "Db Plc <=> HMI".CAGE18_4.DB100_DBX127_00;
      ON    "M186.0";
      =     "M195.5";
END_FUNCTION

FUNCTION "Cage 18 unit" : VOID	// FC 20
TITLE = CAGE 18 UNIT FUNCTION
AUTHOR : Milesi
VERSION : 0.1
VAR_TEMP
  Brake_value : INT ;
END_VAR
BEGIN
NETWORK
TITLE = CAGE 18 OFF
      A(;
      L     "Cage 18".DB20_DBW2;
      L     0;
      ==I;
      );
      AN    "M180.1";
      AN    "M20.0";
      JNB   _001;
      R     "M186.0";
_001: NOP   0;
NETWORK
TITLE = CAGE 18 ON
      A(;
      L     "Cage 18".DB20_DBW2;
      L     1;
      ==I;
      );
      AN    "M180.1";
      AN    "M20.0";
      JNB   _040;
      S     "M186.0";
_040: NOP   0;
NETWORK
TITLE = CAGE 18 Z ROTATION
      A(;
      L     "Cage 18".DB20_DBW4;
      L     0;
      ==I;
      );
      AN    "M180.1";
      AN    "M20.0";
      JNB   _002;
      S     "M186.2";
      R     "M186.3";
_002: NOP   0;
NETWORK
TITLE = CAGE 18 S ROTATION
      A(;
      L     "Cage 18".DB20_DBW4;
      L     1;
      ==I;
      );
      AN    "M180.1";
      AN    "M20.0";
      JNB   _003;
      S     "M186.3";
      R     "M186.2";
_003: NOP   0;
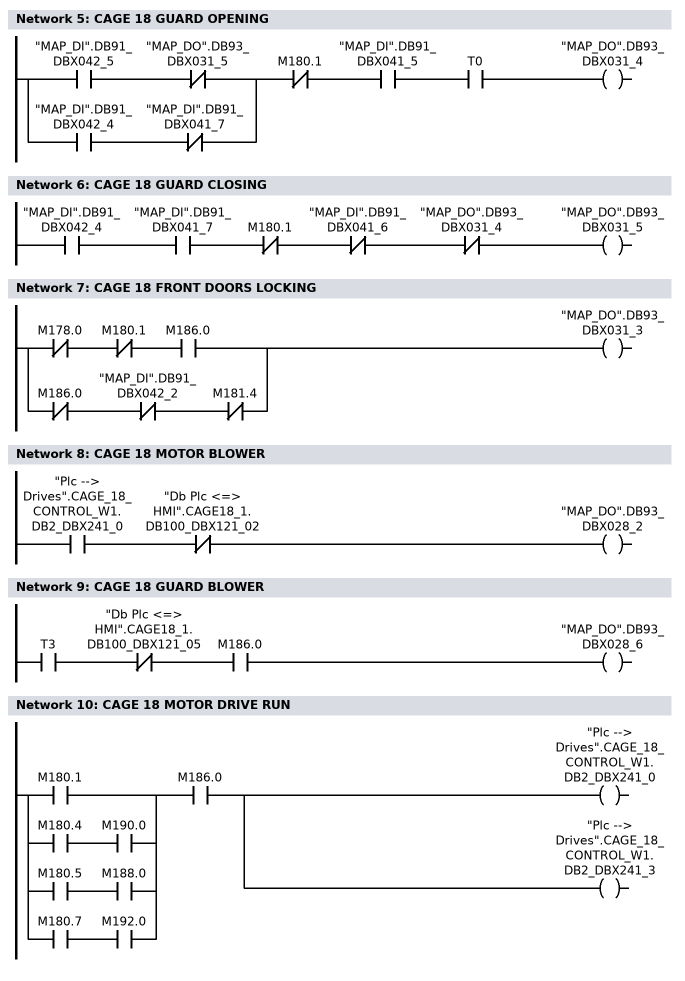
NETWORK
TITLE = CAGE 18 GUARD OPENING
      A(;
      A     "MAP_DI".DB91_DBX042_5;
      AN    "MAP_DO".DB93_DBX031_5;
      O;
      A     "MAP_DI".DB91_DBX042_4;
      AN    "MAP_DI".DB91_DBX041_7;
      );
      AN    "M180.1";
      A     "MAP_DI".DB91_DBX041_5;
      A     "T0";
      =     "MAP_DO".DB93_DBX031_4;
NETWORK
TITLE = CAGE 18 GUARD CLOSING
      A     "MAP_DI".DB91_DBX042_4;
      A     "MAP_DI".DB91_DBX041_7;
//      U     E     56.0
      AN    "M180.1";
      AN    "MAP_DI".DB91_DBX041_6;
      AN    "MAP_DO".DB93_DBX031_4;
      =     "MAP_DO".DB93_DBX031_5;
NETWORK
TITLE = CAGE 18 FRONT DOORS LOCKING
      AN    "M178.0";
      AN    "M180.1";
      A     "M186.0";
      O;
      AN    "M186.0";
      AN    "MAP_DI".DB91_DBX042_2;
      AN    "M181.4";
      =     "MAP_DO".DB93_DBX031_3;
NETWORK
TITLE = CAGE 18 MOTOR BLOWER 
      A     "Plc --> Drives".CAGE_18_CONTROL_W1.DB2_DBX241_0;
      AN    "Db Plc <=> HMI".CAGE18_1.DB100_DBX121_02;
      =     "MAP_DO".DB93_DBX028_2;
NETWORK
TITLE = CAGE 18 GUARD BLOWER
      A     "T3";
      AN    "Db Plc <=> HMI".CAGE18_1.DB100_DBX121_05;
      A     "M186.0";
      =     "MAP_DO".DB93_DBX028_6;
NETWORK
TITLE = CAGE 18 MOTOR DRIVE RUN
      A(;
      O     "M180.1";
      O;
      A     "M180.4";
      A     "M190.0";
      O;
      A     "M180.5";
      A     "M188.0";
      O;
      A     "M180.7";
      A     "M192.0";
      );
      A     "M186.0";
      =     "Plc --> Drives".CAGE_18_CONTROL_W1.DB2_DBX241_0;
      =     "Plc --> Drives".CAGE_18_CONTROL_W1.DB2_DBX241_3;
NETWORK
TITLE = CAGE 18 LAY SET ENABLE
      O     "M180.1";
      O     "M180.6";
      O(;
      A     "M180.4";
      A     "M190.0";
      );
      O(;
      A     "M180.5";
      A     "M188.0";
      );
      O(;
      A     "M180.7";
      A     "M192.0";
      );
      JC    _lay;
      L     "Cage 18".DB20_DBD20;
      T     "Cage 18".DB20_DBD24;
      JU    end1;
_lay: L     "Cage 18".DB20_DBD24;
      T     "Cage 18".DB20_DBD20;
end1: NOP   0;
NETWORK
TITLE = CAGE 18 MOTOR REFERENCE
//Max Linear Speed = 60 m/min
//Max Cage Rpm = 280
//
//Max Linear Speed              60000
//---------------- = Cage Lay = ----- = 214.2
//  Max Cage Rpm                 280
//
//                             Max Linear Speed
//Max Cage Rpm = 280 = 16384 = ---------------- * K
//                                Cage Lay
//
//    Cage Lay * 16384   214.2 * 16384
//K = ---------------- = ------------- = 58490.88
//    Max Linear Speed        60
// (network holds code this reader does not know; not shown)
NETWORK
TITLE = CAGE 18 MAX LINEAR SPEED TO START
      AN    "M200.1";
      JNB   _017;
      L     "Cage 18".DB20_DBD24;
      L     1.750000e-01;
      *R;
      JU    _018;
_017: L     "Cage 18".DB20_DBD24;
      L     2.300000e-01;
      *R;
_018: T     "Cage 18".DB20_DBD120;
      O(;
      L     6.000000e+01;
      >R;
      );
      ON    "M186.0";
      JNB   _014;
      T     "Cage 18".DB20_DBD120;
_014: NOP   0;
NETWORK
TITLE = CAGE 18 MAX LINEAR SPEED
      L     "Cage 18".DB20_DBD24;
      L     2.800000e-01;
      *R;
      T     "Cage 18".DB20_DBD96;
      O(;
      L     6.000000e+01;
      >R;
      );
      ON    "M186.0";
      JNB   _015;
      T     "Cage 18".DB20_DBD96;
_015: NOP   0;
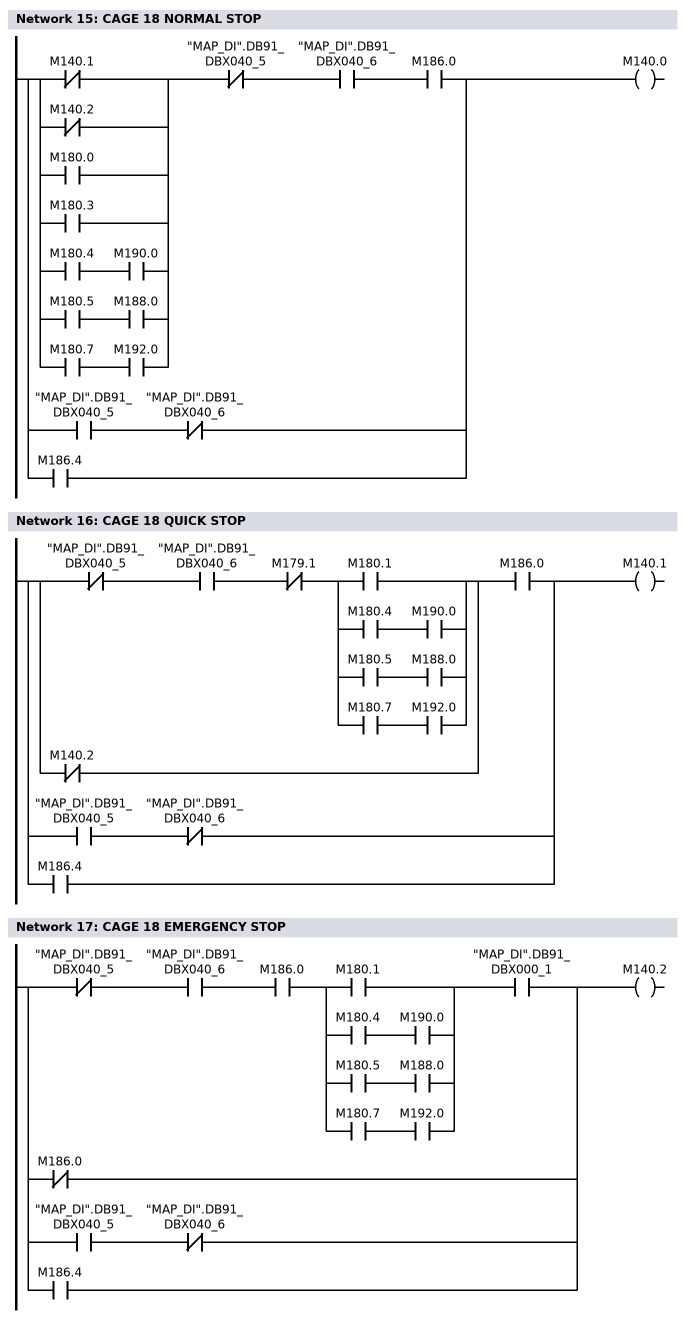
NETWORK
TITLE = CAGE 18 NORMAL STOP
      A(;
      ON    "M140.1";
      ON    "M140.2";
      O     "M180.0";
      O     "M180.3";
      O;
      A     "M180.4";
      A     "M190.0";
      O;
      A     "M180.5";
      A     "M188.0";
      O;
      A     "M180.7";
      A     "M192.0";
      );
      AN    "MAP_DI".DB91_DBX040_5;
      A     "MAP_DI".DB91_DBX040_6;
      A     "M186.0";
      O;
      A     "MAP_DI".DB91_DBX040_5;
      AN    "MAP_DI".DB91_DBX040_6;
      O     "M186.4";
      =     "M140.0";
NETWORK
TITLE = CAGE 18 QUICK STOP
      A(;
      AN    "MAP_DI".DB91_DBX040_5;
      A     "MAP_DI".DB91_DBX040_6;
      AN    "M179.1";
      A(;
      O     "M180.1";
      O;
      A     "M180.4";
      A     "M190.0";
      O;
      A     "M180.5";
      A     "M188.0";
      O;
      A     "M180.7";
      A     "M192.0";
      );
      ON    "M140.2";
      );
      A     "M186.0";
      O;
      A     "MAP_DI".DB91_DBX040_5;
      AN    "MAP_DI".DB91_DBX040_6;
      O     "M186.4";
      =     "M140.1";
NETWORK
TITLE = CAGE 18 EMERGENCY STOP
      AN    "MAP_DI".DB91_DBX040_5;
      A     "MAP_DI".DB91_DBX040_6;
      A     "M186.0";
      A(;
      O     "M180.1";
      O;
      A     "M180.4";
      A     "M190.0";
      O;
      A     "M180.5";
      A     "M188.0";
      O;
      A     "M180.7";
      A     "M192.0";
      );
      A     "MAP_DI".DB91_DBX000_1;
      ON    "M186.0";
      O;
      A     "MAP_DI".DB91_DBX040_5;
      AN    "MAP_DI".DB91_DBX040_6;
      O     "M186.4";
      =     "M140.2";
NETWORK
TITLE = CAGE 18 BRAKE PROPORTIONAL VALVE REFERENCE
      A     "M140.0";
      JC    _004;
      L     "Cage 18".DB20_DBD64;
      L     1.000000e+02;
      /R;
      L     2.764800e+04;
      *R;
      RND;
      JU    BRK;
_004: A     "M140.1";
      JC    _005;
      L     "Cage 18".DB20_DBD68;
      L     1.000000e+02;
      /R;
      L     2.764800e+04;
      *R;
      RND;
      JU    BRK;
_005: A     "M140.2";
      JC    _006;
      L     "Cage 18".DB20_DBD72;
      L     1.000000e+02;
      /R;
      L     2.764800e+04;
      *R;
      RND;
      JU    BRK;
_006: L     0;
BRK:  T     #Brake_value;
NETWORK
TITLE = SET POINT IN AMPER CALCULATION
      L     "Cage 18".DB20_DBD276;
      L     1.600000e+02;
      *R;
      L     1.000000e+02;
      /R;
      T     "Cage 18".DB20_DBD260;
NETWORK
TITLE = CURRENT CALCULATION
// (network holds code this reader does not know; not shown)
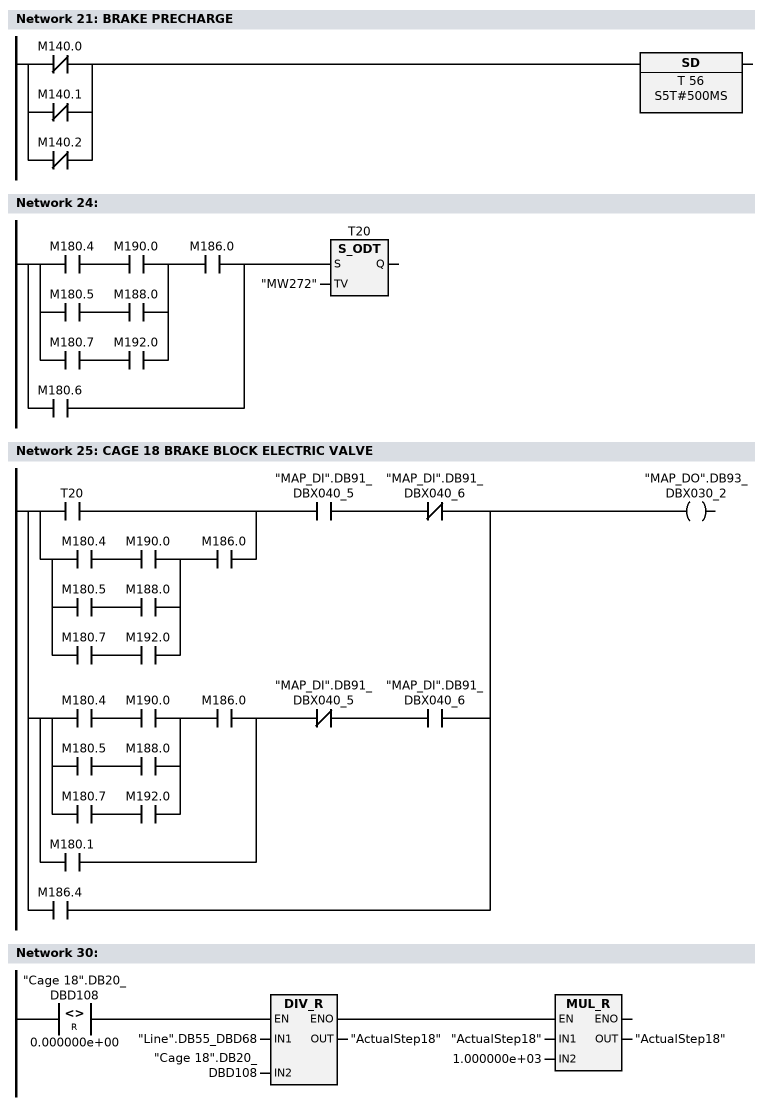
NETWORK
TITLE = BRAKE PRECHARGE
      ON    "M140.0";
      ON    "M140.1";
      ON    "M140.2";
      L     S5T#500MS;
      SD    T 56;
NETWORK
TITLE = BRAKE MODULATION CONTROL
      L     "Cage 18".DB20_DBD260;
      L     "Cage 18".DB20_DBD200;
      -R;
      T     "Cage 18".DB20_DBD264;
      L     "Cage 18".DB20_DBD268;
      *R;
      T     "Cage 18".DB20_DBD272;
      L     2.768400e+04;
      >R;
      JCN   _20d;
      L     2.768400e+04;
      T     "Cage 18".DB20_DBD272;
_20d: A     T 56;
      A     "M180.1";
      JCN   _20b;
      A(;
      L     "Cage 18".DB20_DBD272;
      L     0.000000e+00;
      <R;
      );
      JCN   _20a;
      L     0.000000e+00;
      T     "Cage 18".DB20_DBD272;
_20a: L     "Cage 18".DB20_DBD272;
      RND;
      JU    _20c;
_20b: L     #Brake_value;
_20c: T     "-559Y1";
NETWORK
TITLE = CAGE 18 BRAKE BLOCK OPEN ON-DELAY TIMER
      L     "Cage 18".DB20_DBD148;
      RND;
      ITB;
      L     W#16#2000;
      OW;
      T     "MW272";
NETWORK
TITLE =
      A(;
      A(;
      A     "M180.4";
      A     "M190.0";
      O;
      A     "M180.5";
      A     "M188.0";
      O;
      A     "M180.7";
      A     "M192.0";
      );
      A     "M186.0";
      O     "M180.6";
      );
      L     "MW272";
      SD    "T20";
      NOP   0;
      NOP   0;
      NOP   0;
      NOP   0;
NETWORK
TITLE = CAGE 18 BRAKE BLOCK ELECTRIC VALVE
      A(;
      O     "T20";
      O;
      A(;
      A     "M180.4";
      A     "M190.0";
      O;
      A     "M180.5";
      A     "M188.0";
      O;
      A     "M180.7";
      A     "M192.0";
      );
      A     "M186.0";
      );
      A     "MAP_DI".DB91_DBX040_5;
      AN    "MAP_DI".DB91_DBX040_6;
      O;
      A(;
      A(;
      A     "M180.4";
      A     "M190.0";
      O;
      A     "M180.5";
      A     "M188.0";
      O;
      A     "M180.7";
      A     "M192.0";
      );
      A     "M186.0";
      O     "M180.1";
      );
      AN    "MAP_DI".DB91_DBX040_5;
      A     "MAP_DI".DB91_DBX040_6;
      O     "M186.4";
      =     "MAP_DO".DB93_DBX030_2;
NETWORK
TITLE = CAGE 18 RPM TO HMI
      L     "Drives --> Plc".DB1_DBW246;
      ITD;
      DTR;
      L     1.638400e+04;
      /R;
      L     2.800000e+02;
      *R;
      ABS;
      T     "Cage 18".DB20_DBD108;
NETWORK
TITLE = CAGE 18 MOTOR RPM TO HMI
      L     "Drives --> Plc".DB1_DBW246;
      ITD;
      DTR;
      L     1.638400e+04;
      /R;
      L     1.460000e+03;
      *R;
      T     "Cage 18".DB20_DBD188;
NETWORK
TITLE = CAGE 18 MOTOR CURRENT TO HMI
      L     "Drives --> Plc".DB1_DBW248;
      ITD;
      DTR;
      L     1.638400e+04;
      /R;
      L     1.600000e+02;
      *R;
      T     "Cage 18".DB20_DBD192;
NETWORK
TITLE = CAGE 18 MOTOR VOLTAGE TO HMI
      L     "Drives --> Plc".DB1_DBW250;
      ITD;
      DTR;
      L     1.638400e+04;
      /R;
      L     4.000000e+02;
      *R;
      T     "Cage 18".DB20_DBD196;
NETWORK
TITLE =
      A(;
      A(;
      L     "Cage 18".DB20_DBD108;
      L     0.000000e+00;
      <>R;
      );
      JNB   _007;
      L     "Line".DB55_DBD68;
      L     "Cage 18".DB20_DBD108;
      /R;
      T     "ActualStep18";
      AN    OV;
      SAVE;
      CLR;
_007: A     BR;
      );
      JNB   _008;
      L     "ActualStep18";
      L     1.000000e+03;
      *R;
      T     "ActualStep18";
_008: NOP   0;
END_FUNCTION

FUNCTION "Cage 18 loading fase" : VOID	// FC 21
TITLE = CAGE 18 LOADING FASE FUNCTION
AUTHOR : Milesi
VERSION : 0.1
BEGIN
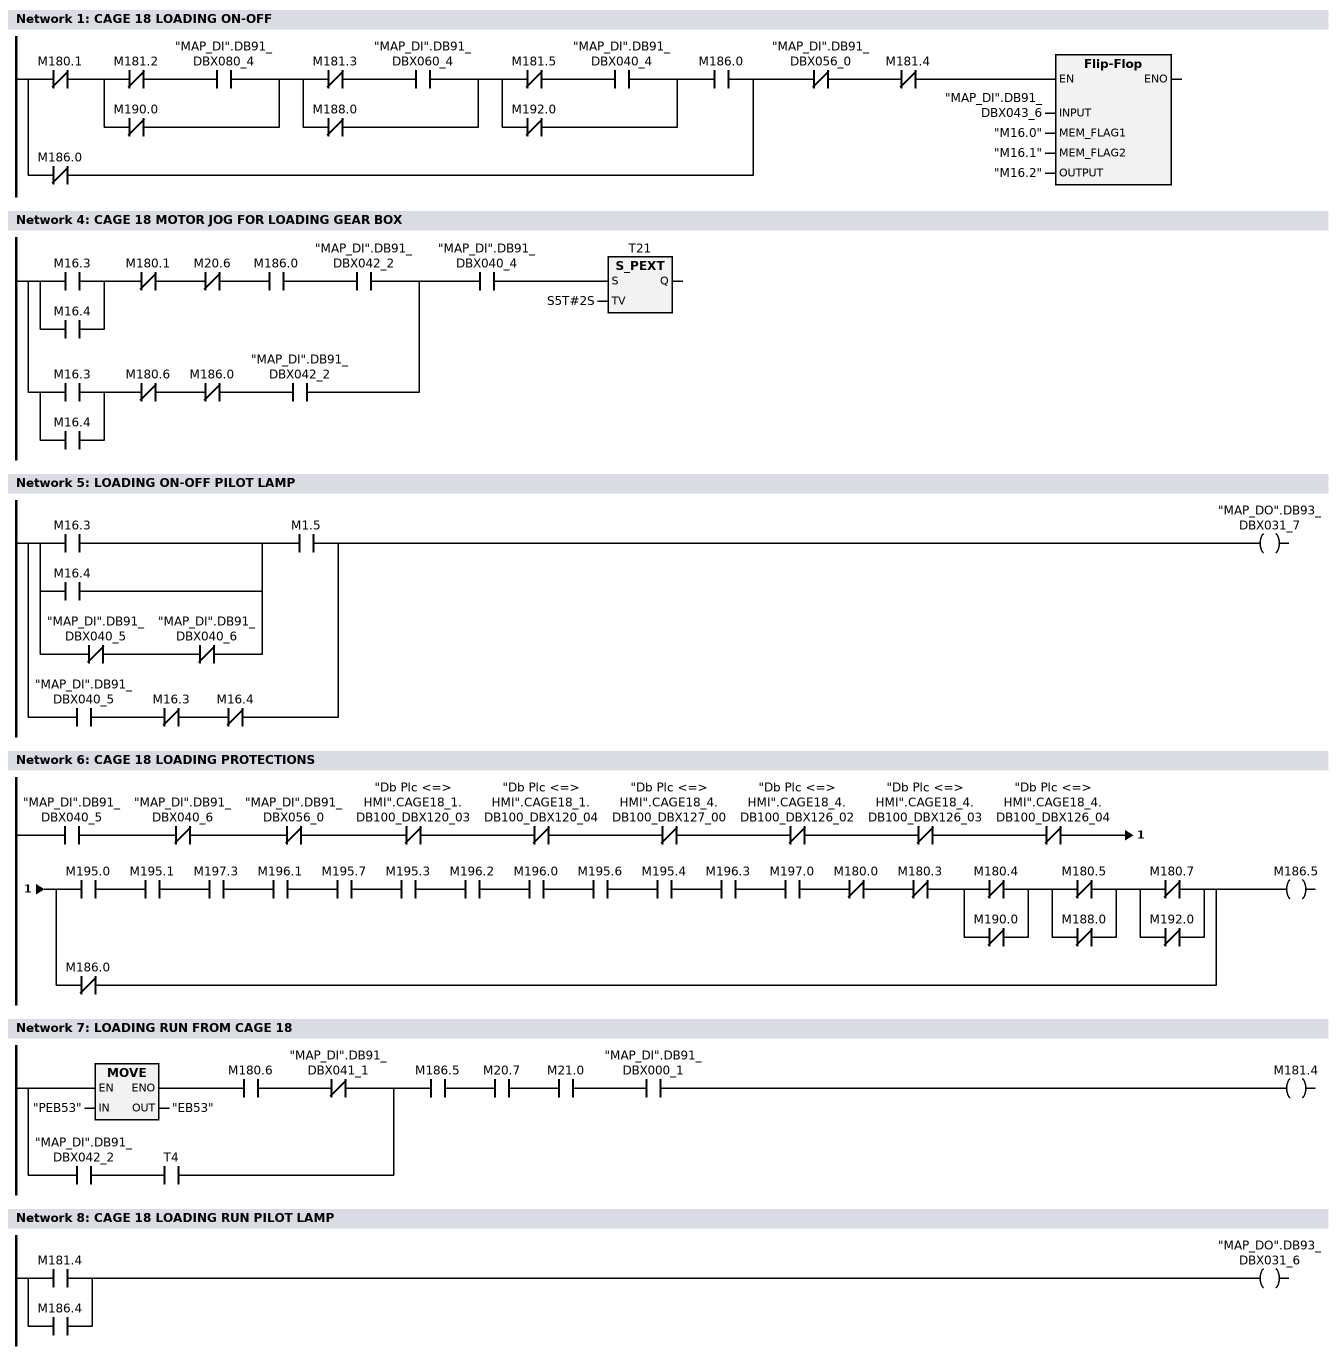
NETWORK
TITLE = CAGE 18 LOADING ON-OFF
      A(;
      AN    "M180.1";
      A(;
      AN    "M181.2";
      A     "MAP_DI".DB91_DBX080_4;
      ON    "M190.0";
      );
      A(;
      AN    "M181.3";
      A     "MAP_DI".DB91_DBX060_4;
      ON    "M188.0";
      );
      A(;
      AN    "M181.5";
      A     "MAP_DI".DB91_DBX040_4;
      ON    "M192.0";
      );
      A     "M186.0";
      ON    "M186.0";
      );
      AN    "MAP_DI".DB91_DBX056_0;
      AN    "M181.4";
      JNB   _001;
      CALL  "Flip-Flop" (
           INPUT                    := "MAP_DI".DB91_DBX043_6,
           MEM_FLAG1                := "M16.0",
           MEM_FLAG2                := "M16.1",
           OUTPUT                   := "M16.2");
_001: NOP   0;
NETWORK
TITLE = CAGE 18 LOADING ON
      A(;
      A(;
      A     "M16.2";
      AN    "M180.1";
      AN    "M20.6";
      A     "M186.0";
      O;
      AN    "M180.6";
      AN    "M186.0";
      );
      S     "MAP_DO".DB93_DBX030_0;
      A(;
      O     "MAP_DI".DB91_DBX040_5;
      O     "MAP_DO".DB93_DBX030_1;
      ON    "M16.2";
      );
      R     "MAP_DO".DB93_DBX030_0;
      A     "MAP_DO".DB93_DBX030_0;
      );
      S     "M16.3";
      A(;
      O     "MAP_DI".DB91_DBX040_5;
      ON    "M16.2";
      );
      R     "M16.3";
      NOP   0;
NETWORK
TITLE = CAGE 18 LOADING OFF
      A(;
      A(;
      AN    "M16.2";
      AN    "M20.6";
      A     "M186.0";
      O;
      AN    "M180.6";
      AN    "M186.0";
      );
      S     "MAP_DO".DB93_DBX030_1;
      A(;
      O     "MAP_DI".DB91_DBX040_6;
      O     "MAP_DO".DB93_DBX030_0;
      O     "M16.2";
      );
      R     "MAP_DO".DB93_DBX030_1;
      A     "MAP_DO".DB93_DBX030_1;
      );
      S     "M16.4";
      A(;
      O     "MAP_DI".DB91_DBX040_6;
      O     "M16.2";
      );
      R     "M16.4";
      NOP   0;
NETWORK
TITLE = CAGE 18 MOTOR JOG FOR LOADING GEAR BOX
      A(;
      A(;
      O     "M16.3";
      O     "M16.4";
      );
      AN    "M180.1";
      AN    "M20.6";
      A     "M186.0";
      A     "MAP_DI".DB91_DBX042_2;
      O;
      A(;
      O     "M16.3";
      O     "M16.4";
      );
      AN    "M180.6";
      AN    "M186.0";
      A     "MAP_DI".DB91_DBX042_2;
      );
      A     "MAP_DI".DB91_DBX040_4;
      L     S5T#2S;
      SE    "T21";
      NOP   0;
      NOP   0;
      NOP   0;
      NOP   0;
NETWORK
TITLE = LOADING ON-OFF PILOT LAMP
      A(;
      O     "M16.3";
      O     "M16.4";
      O;
      AN    "MAP_DI".DB91_DBX040_5;
      AN    "MAP_DI".DB91_DBX040_6;
      );
      A     "M1.5";
      O;
      A     "MAP_DI".DB91_DBX040_5;
      AN    "M16.3";
      AN    "M16.4";
      =     "MAP_DO".DB93_DBX031_7;
NETWORK
TITLE = CAGE 18 LOADING PROTECTIONS
      A     "MAP_DI".DB91_DBX040_5;
      AN    "MAP_DI".DB91_DBX040_6;
      AN    "MAP_DI".DB91_DBX056_0;
      AN    "Db Plc <=> HMI".CAGE18_1.DB100_DBX120_03;
      AN    "Db Plc <=> HMI".CAGE18_1.DB100_DBX120_04;
      AN    "Db Plc <=> HMI".CAGE18_4.DB100_DBX127_00;
      AN    "Db Plc <=> HMI".CAGE18_4.DB100_DBX126_02;
      AN    "Db Plc <=> HMI".CAGE18_4.DB100_DBX126_03;
      AN    "Db Plc <=> HMI".CAGE18_4.DB100_DBX126_04;
      A(;
      A     "M195.0";
      A     "M195.1";
      A     "M197.3";
      A     "M196.1";
      A     "M195.7";
      A     "M195.3";
      A     "M196.2";
      A     "M196.0";
      A     "M195.6";
      A     "M195.4";
      A     "M196.3";
      A     "M197.0";
      AN    "M180.0";
      AN    "M180.3";
      A(;
      ON    "M180.4";
      ON    "M190.0";
      );
      A(;
      ON    "M180.5";
      ON    "M188.0";
      );
      A(;
      ON    "M180.7";
      ON    "M192.0";
      );
      ON    "M186.0";
      );
      =     "M186.5";
NETWORK
TITLE = LOADING RUN FROM CAGE 18
      A(;
      A(;
      L     "PEB53";
      T     "EB53";
      SET;
      SAVE;
      CLR;
      A     BR;
      );
      A     "M180.6";
      AN    "MAP_DI".DB91_DBX041_1;
      O;
      A     "MAP_DI".DB91_DBX042_2;
      A     "T4";
      );
      A     "M186.5";
      A     "M20.7";
      A     "M21.0";
      A     "MAP_DI".DB91_DBX000_1;
      =     "M181.4";
NETWORK
TITLE = CAGE 18 LOADING RUN PILOT LAMP
      O     "M181.4";
      O     "M186.4";
      =     "MAP_DO".DB93_DBX031_6;
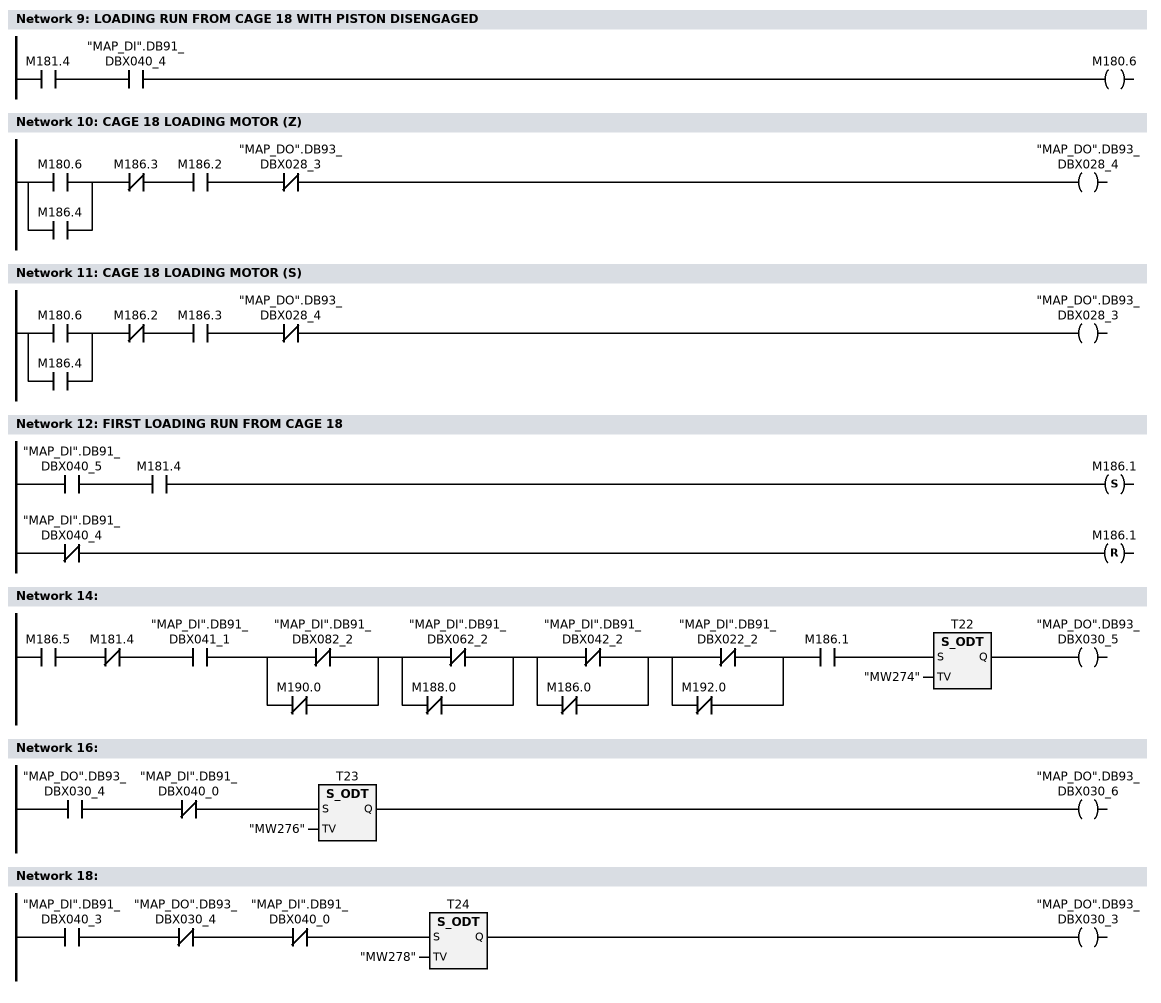
NETWORK
TITLE = LOADING RUN FROM CAGE 18 WITH PISTON DISENGAGED
      A     "M181.4";
      A     "MAP_DI".DB91_DBX040_4;
      =     "M180.6";
NETWORK
TITLE = CAGE 18 LOADING MOTOR (Z)
      A(;
      O     "M180.6";
      O     "M186.4";
      );
      AN    "M186.3";
      A     "M186.2";
      AN    "MAP_DO".DB93_DBX028_3;
      =     "MAP_DO".DB93_DBX028_4;
NETWORK
TITLE = CAGE 18 LOADING MOTOR (S)
      A(;
      O     "M180.6";
      O     "M186.4";
      );
      AN    "M186.2";
      A     "M186.3";
      AN    "MAP_DO".DB93_DBX028_4;
      =     "MAP_DO".DB93_DBX028_3;
NETWORK
TITLE = FIRST LOADING RUN FROM CAGE 18
      A     "MAP_DI".DB91_DBX040_5;
      A     "M181.4";
      S     "M186.1";
      AN    "MAP_DI".DB91_DBX040_4;
      R     "M186.1";
      NOP   0;
NETWORK
TITLE = CAGE 18 PISTON ENGAGING INTO CAGE
      L     "Cage 18".DB20_DBD152;
      RND;
      ITB;
      L     W#16#2000;
      OW;
      T     "MW274";
NETWORK
TITLE =
      A     "M186.5";
      AN    "M181.4";
      A     "MAP_DI".DB91_DBX041_1;
      A(;
      ON    "MAP_DI".DB91_DBX082_2;
      ON    "M190.0";
      );
      A(;
      ON    "MAP_DI".DB91_DBX062_2;
      ON    "M188.0";
      );
      A(;
      ON    "MAP_DI".DB91_DBX042_2;
      ON    "M186.0";
      );
      A(;
      ON    "MAP_DI".DB91_DBX022_2;
      ON    "M192.0";
      );
      A     "M186.1";
      L     "MW274";
      SD    "T22";
      NOP   0;
      NOP   0;
      NOP   0;
      A     "T22";
      =     "MAP_DO".DB93_DBX030_5;
NETWORK
TITLE = CAGE 18 PISTON DISENGAGING FROM CAGE
      L     "Cage 18".DB20_DBD144;
      RND;
      ITB;
      L     W#16#2000;
      OW;
      T     "MW276";
NETWORK
TITLE =
      A     "MAP_DO".DB93_DBX030_4;
      AN    "MAP_DI".DB91_DBX040_0;
      L     "MW276";
      SD    "T23";
      NOP   0;
      NOP   0;
      NOP   0;
      A     "T23";
      =     "MAP_DO".DB93_DBX030_6;
NETWORK
TITLE = CAGE 18 AIR INLET INTO CAGE
      L     "Cage 18".DB20_DBD156;
      RND;
      ITB;
      L     W#16#2000;
      OW;
      T     "MW278";
NETWORK
TITLE =
      A     "MAP_DI".DB91_DBX040_3;
      AN    "MAP_DO".DB93_DBX030_4;
      AN    "MAP_DI".DB91_DBX040_0;
      L     "MW278";
      SD    "T24";
      NOP   0;
      NOP   0;
      NOP   0;
      A     "T24";
      =     "MAP_DO".DB93_DBX030_3;
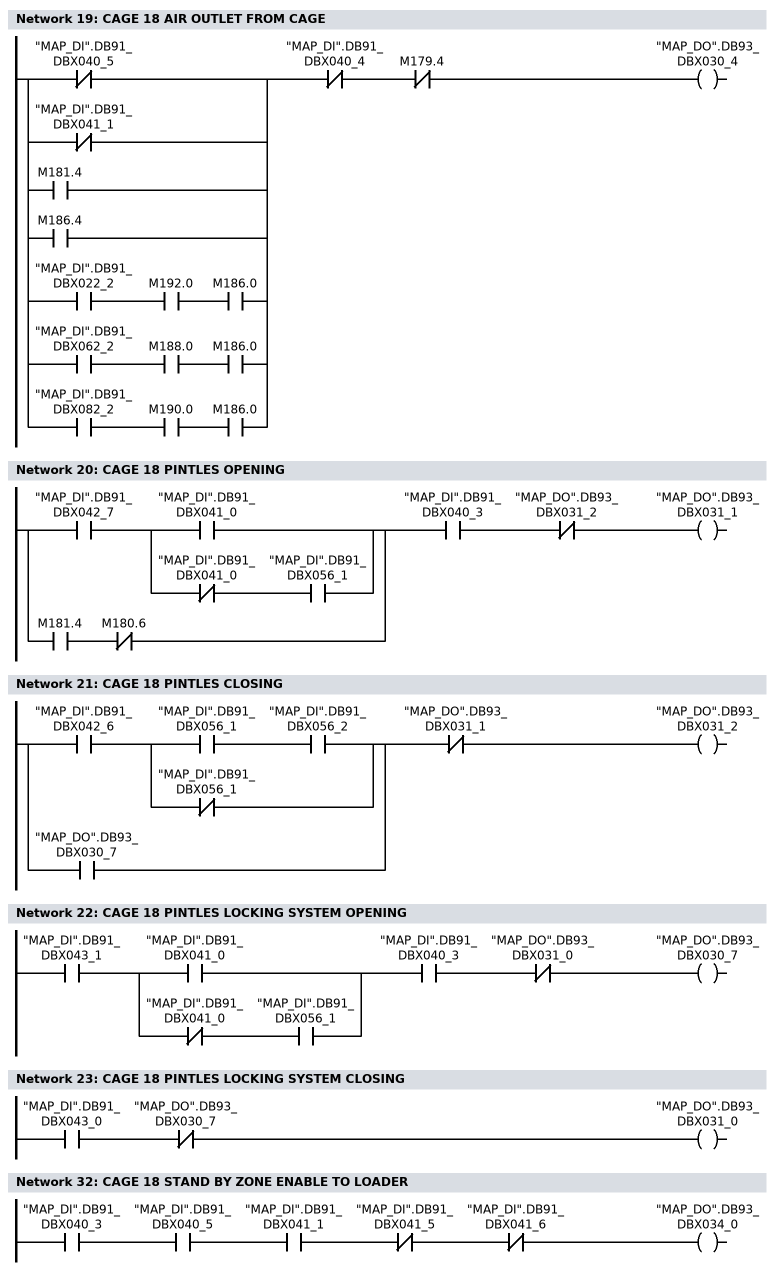
NETWORK
TITLE = CAGE 18 AIR OUTLET FROM CAGE
      A(;
      ON    "MAP_DI".DB91_DBX040_5;
      ON    "MAP_DI".DB91_DBX041_1;
      O     "M181.4";
      O     "M186.4";
      O;
      A     "MAP_DI".DB91_DBX022_2;
      A     "M192.0";
      A     "M186.0";
      O;
      A     "MAP_DI".DB91_DBX062_2;
      A     "M188.0";
      A     "M186.0";
      O;
      A     "MAP_DI".DB91_DBX082_2;
      A     "M190.0";
      A     "M186.0";
      );
      AN    "MAP_DI".DB91_DBX040_4;
      AN    "M179.4";
      =     "MAP_DO".DB93_DBX030_4;
NETWORK
TITLE = CAGE 18 PINTLES OPENING
      A(;
      A     "MAP_DI".DB91_DBX042_7;
      A(;
      O     "MAP_DI".DB91_DBX041_0;
      O;
      AN    "MAP_DI".DB91_DBX041_0;
      A     "MAP_DI".DB91_DBX056_1;
      );
      O;
      A     "M181.4";
      AN    "M180.6";
      );
      A     "MAP_DI".DB91_DBX040_3;
      AN    "MAP_DO".DB93_DBX031_2;
      =     "MAP_DO".DB93_DBX031_1;
NETWORK
TITLE = CAGE 18 PINTLES CLOSING
      A(;
      A     "MAP_DI".DB91_DBX042_6;
      A(;
      A     "MAP_DI".DB91_DBX056_1;
      A     "MAP_DI".DB91_DBX056_2;
      ON    "MAP_DI".DB91_DBX056_1;
      );
      O     "MAP_DO".DB93_DBX030_7;
      );
      AN    "MAP_DO".DB93_DBX031_1;
      =     "MAP_DO".DB93_DBX031_2;
NETWORK
TITLE = CAGE 18 PINTLES LOCKING SYSTEM OPENING
      A     "MAP_DI".DB91_DBX043_1;
      A(;
      O     "MAP_DI".DB91_DBX041_0;
      O;
      AN    "MAP_DI".DB91_DBX041_0;
      A     "MAP_DI".DB91_DBX056_1;
      );
      A     "MAP_DI".DB91_DBX040_3;
      AN    "MAP_DO".DB93_DBX031_0;
      =     "MAP_DO".DB93_DBX030_7;
NETWORK
TITLE = CAGE 18 PINTLES LOCKING SYSTEM CLOSING
      A     "MAP_DI".DB91_DBX043_0;
      AN    "MAP_DO".DB93_DBX030_7;
      =     "MAP_DO".DB93_DBX031_0;
NETWORK
TITLE = CAGE 18 PLATFORM UP
NETWORK
TITLE = CAGE 18 PLATFORM DOWN
NETWORK
TITLE = CAGE 18 EVEN BOBBINS ROTATION FOR LOADING MACHINE
NETWORK
TITLE = CAGE 18 EVEN BOBBINS ROTATION FOR LOADING PLATFORM
NETWORK
TITLE = CAGE 18 ODD BOBBINS ROTATION FOR LOADING MACHINE
NETWORK
TITLE = CAGE 18 ODD BOBBINS ROTATION FOR LOADING PLATFORM
NETWORK
TITLE = CAGE 18 BOBBIN ROTATION FOR LOADING MACHINE PILOT LAMP
NETWORK
TITLE = CAGE 18 LOADING PUMP
NETWORK
TITLE = CAGE 18 STAND BY ZONE ENABLE TO LOADER
      A     "MAP_DI".DB91_DBX040_3;
      A     "MAP_DI".DB91_DBX040_5;
      A     "MAP_DI".DB91_DBX041_1;
      AN    "MAP_DI".DB91_DBX041_5;
      AN    "MAP_DI".DB91_DBX041_6;
      =     "MAP_DO".DB93_DBX034_0;
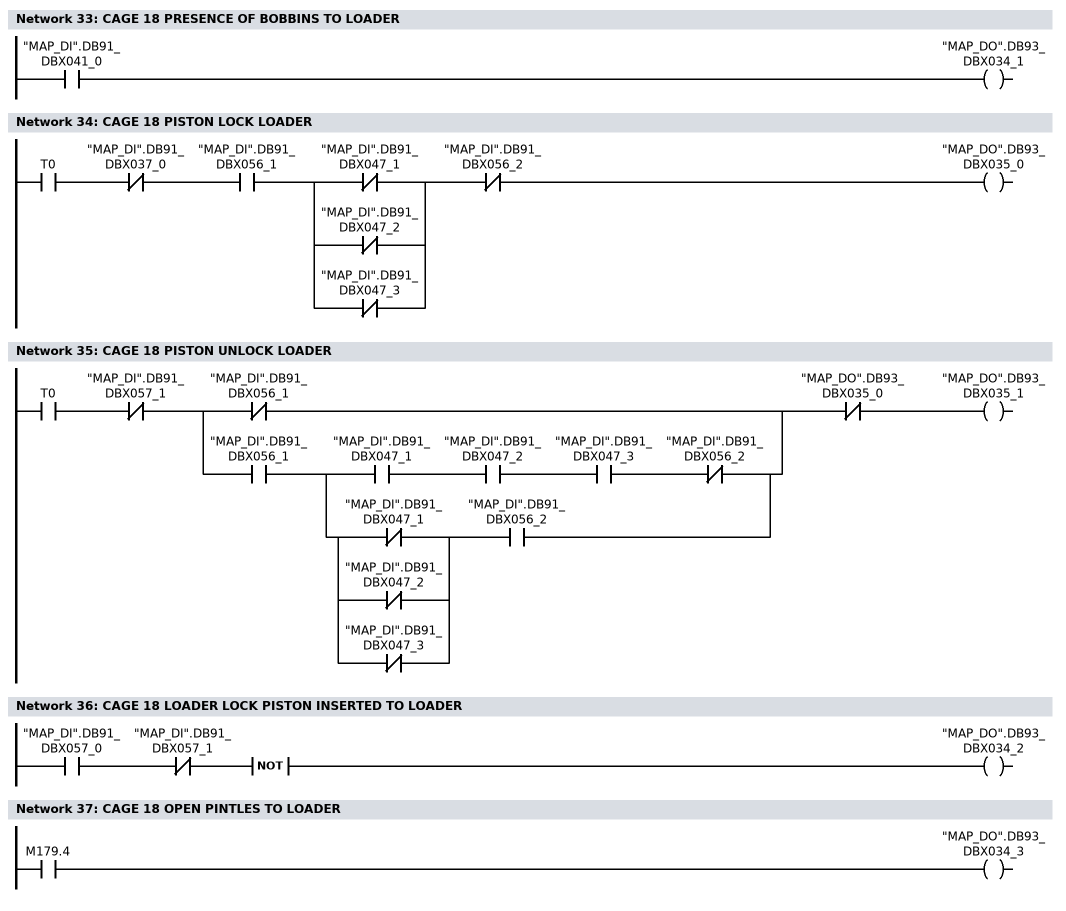
NETWORK
TITLE = CAGE 18 PRESENCE OF BOBBINS TO LOADER
      A     "MAP_DI".DB91_DBX041_0;
      =     "MAP_DO".DB93_DBX034_1;
NETWORK
TITLE = CAGE 18 PISTON LOCK LOADER
      A     "T0";
      AN    "MAP_DI".DB91_DBX037_0;
      A     "MAP_DI".DB91_DBX056_1;
      A(;
      ON    "MAP_DI".DB91_DBX047_1;
      ON    "MAP_DI".DB91_DBX047_2;
      ON    "MAP_DI".DB91_DBX047_3;
      );
      AN    "MAP_DI".DB91_DBX056_2;
      =     "MAP_DO".DB93_DBX035_0;
NETWORK
TITLE = CAGE 18 PISTON UNLOCK LOADER
      A     "T0";
      AN    "MAP_DI".DB91_DBX057_1;
      A(;
      ON    "MAP_DI".DB91_DBX056_1;
      O;
      A     "MAP_DI".DB91_DBX056_1;
      A(;
      A     "MAP_DI".DB91_DBX047_1;
      A     "MAP_DI".DB91_DBX047_2;
      A     "MAP_DI".DB91_DBX047_3;
      AN    "MAP_DI".DB91_DBX056_2;
      O;
      A(;
      ON    "MAP_DI".DB91_DBX047_1;
      ON    "MAP_DI".DB91_DBX047_2;
      ON    "MAP_DI".DB91_DBX047_3;
      );
      A     "MAP_DI".DB91_DBX056_2;
      );
      );
      AN    "MAP_DO".DB93_DBX035_0;
      =     "MAP_DO".DB93_DBX035_1;
NETWORK
TITLE = CAGE 18 LOADER LOCK PISTON INSERTED TO LOADER 
      A     "MAP_DI".DB91_DBX057_0;
      AN    "MAP_DI".DB91_DBX057_1;
      NOT;
      =     "MAP_DO".DB93_DBX034_2;
NETWORK
TITLE = CAGE 18 OPEN PINTLES TO LOADER
      A     "M179.4";
      =     "MAP_DO".DB93_DBX034_3;
END_FUNCTION

FUNCTION "Cage 18 preforming alarm" : VOID	// FC 22
TITLE = CAGE 18 PREFORMING ALARMS FUNCTION
AUTHOR : Milesi
VERSION : 0.1
BEGIN
NETWORK
TITLE = CAGE 18 PREFORMING MOTOR DRIVE PROFIBUS SLAVE 8 FAULT
      A(;
      L     "MB304";
      L     8;
      ==I;
      );
      AN    "M300.5";
      S     "Db Plc <=> HMI".PROFIBUS.DB100_DBX101_7;
NETWORK
TITLE = CAGE 18 PREFORMING MOTOR BRAKE OVERLOAD
      A     "T0";
      A     "MAP_DI".DB91_DBX038_4;
      A     "M187.3";
      =     "Db Plc <=> HMI".CAGE18_4.DB100_DBX127_04;
NETWORK
TITLE = CAGE 18 PREFORMING MOTOR BLOWER OVERLOAD
      A     "T0";
      A     "MAP_DI".DB91_DBX038_5;
      A     "M187.3";
      =     "Db Plc <=> HMI".CAGE18_4.DB100_DBX127_05;
NETWORK
TITLE = CAGE 18 PREFORMING OPEN GUARD
      A     "T0";
      A     "M180.1";
      AN    "MAP_DI".DB91_DBX044_6;
      A     "M187.3";
      S     "M174.4";
NETWORK
TITLE =
      A     "T0";
      A(;
      ON    "MAP_DI".DB91_DBX044_6;
      O     "M174.4";
      );
      A     "M187.3";
      =     "Db Plc <=> HMI".CAGE18_4.DB100_DBX127_06;
NETWORK
TITLE = CAGE 18 PREFORMING MOTOR DRIVE FAULT
      A     "T0";
      A     "Drives --> Plc".CAGE_18_PREF_STATUS_W1.DB1_DBX201_3;
      A     "M187.3";
      S     "Db Plc <=> HMI".CAGE18_4.DB100_DBX127_07;
NETWORK
TITLE = CAGE 18 PREFORMING GENERAL ALARM
      AN    "Db Plc <=> HMI".PROFIBUS.DB100_DBX101_7;
      AN    "Db Plc <=> HMI".CAGE18_4.DB100_DBX127_04;
      AN    "Db Plc <=> HMI".CAGE18_4.DB100_DBX127_05;
      AN    "Db Plc <=> HMI".CAGE18_4.DB100_DBX127_06;
      AN    "Db Plc <=> HMI".CAGE18_4.DB100_DBX127_07;
      =     "M195.6";
END_FUNCTION

FUNCTION "Cage 18 preforming unit" : VOID	// FC 23
TITLE = CAGE 18 PREFORMING UNIT FUNCTION
AUTHOR : Milesi
VERSION : 0.1
BEGIN
NETWORK
TITLE = CAGE 18 PREFORMING OFF
      A(;
      L     "Cage 18 preforming".DB23_DBW2;
      L     0;
      ==I;
      );
      AN    "M180.1";
      JNB   _001;
      R     "M187.3";
      R     "M187.4";
      R     "M187.5";
_001: NOP   0;
NETWORK
TITLE = CAGE 18 PREFORMING Z ROTATION
      A(;
      L     "Cage 18 preforming".DB23_DBW2;
      L     1;
      ==I;
      );
      AN    "M180.1";
      JNB   _002;
      S     "M187.3";
      S     "M187.4";
      R     "M187.5";
_002: NOP   0;
NETWORK
TITLE = CAGE 18 PREFORMING S ROTATION
      A(;
      L     "Cage 18 preforming".DB23_DBW2;
      L     2;
      ==I;
      );
      AN    "M180.1";
      JNB   _003;
      S     "M187.3";
      S     "M187.5";
      R     "M187.4";
_003: NOP   0;
NETWORK
TITLE = CAGE 18 PREFORMING MOTOR DRIVE RUN
      A(;
      O     "M180.1";
      O     "M21.3";
      );
      AN    "Db Plc <=> HMI".CAGE18_4.DB100_DBX127_07;
      A     "M187.3";
      =     "Plc --> Drives".CAGE_18_PREF_CONTROL_W1.DB2_DBX201_0;
      =     "Plc --> Drives".CAGE_18_PREF_CONTROL_W1.DB2_DBX201_3;
NETWORK
TITLE = CAGE 18 PREFORMING MOTOR BLOWER
      A     "Plc --> Drives".CAGE_18_PREF_CONTROL_W1.DB2_DBX201_0;
      AN    "Db Plc <=> HMI".CAGE18_4.DB100_DBX127_05;
      =     "MAP_DO".DB93_DBX028_1;
NETWORK
TITLE = CAGE 18 PREFORMING MOTOR ELECTRIC BRAKE RELAY
      A(;
      O     "Plc --> Drives".CAGE_18_PREF_CONTROL_W1.DB2_DBX201_0;
      O     "MAP_DI".DB91_DBX044_7;
      );
      AN    "Db Plc <=> HMI".CAGE18_4.DB100_DBX127_05;
      =     "MAP_DO".DB93_DBX028_0;
NETWORK
TITLE = CAGE 18 PREFORMING MOTOR REFERENCE
//Max Linear Speed = 40 m/min
//Max Die Rpm = 147.68
//
//Max Linear Speed             40000
//---------------- = Die Lay = ------ = 270.85
//  Max Die Rpm                147.68
//
//                               Max Linear Speed
//Max Die Rpm = 147.68 = 16384 = ---------------- * K
//                                   Die Lay
//
//    Die Lay * 16384   270.85 * 16384
//K = ---------------- = ------------- = 110940.16
//    Max Linear Speed        40
// (network holds code this reader does not know; not shown)
NETWORK
TITLE = CAGE 18 PREFORMING RPM TO HMI
      L     "Drives --> Plc".DB1_DBW206;
      ITD;
      DTR;
      L     1.638400e+04;
      /R;
      L     1.476800e+02;
      *R;
      ABS;
      T     "Cage 18 preforming".DB23_DBD108;
NETWORK
TITLE = CAGE 18 PREFORMING MOTOR RPM TO HMI
      L     "Drives --> Plc".DB1_DBW206;
      ITD;
      DTR;
      L     1.638400e+04;
      /R;
      L     1.420000e+03;
      *R;
      T     "Cage 18 preforming".DB23_DBD188;
NETWORK
TITLE = CAGE 18 PREFORMING MOTOR CURRENT TO HMI
//TORQUE FEEDBACK = 150% = MOTOR CURRENT * 1.5
      L     "Drives --> Plc".DB1_DBW208;
      ITD;
      DTR;
      L     1.638400e+04;
      /R;
      L     3.400000e+00;
      *R;
      T     "Cage 18 preforming".DB23_DBD192;
NETWORK
TITLE = CAGE 18 PREFORMING MOTOR VOLTAGE TO HMI
      L     "Drives --> Plc".DB1_DBW210;
      ITD;
      DTR;
      L     1.638400e+04;
      /R;
      L     4.000000e+02;
      *R;
      T     "Cage 18 preforming".DB23_DBD196;
END_FUNCTION

FUNCTION "Cage 12 alarms" : VOID	// FC 24
TITLE = CAGE 12 ALARMS FUNCTION
AUTHOR : Milesi
VERSION : 0.1
VAR_TEMP
  T4_time : WORD ;
END_VAR
BEGIN
NETWORK
TITLE = CAGE 12 MOTOR DRIVE PROFIBUS SLAVE 11 FAULT
      A(;
      L     "MB304";
      L     11;
      ==I;
      );
      AN    "M300.5";
      S     "Db Plc <=> HMI".PROFIBUS.DB100_DBX100_2;
NETWORK
TITLE = CAGE 12 ET200M PROFIBUS SLAVE 23 FAULT
      A(;
      L     "MB304";
      L     23;
      ==I;
      );
      AN    "M300.5";
      S     "Db Plc <=> HMI".PROFIBUS.DB100_DBX100_7;
NETWORK
TITLE = CAGE 12 OPEN FRONT GUARD
      A     "T0";
      A     "M180.1";
      AN    "MAP_DI".DB91_DBX061_6;
      A     "M188.0";
      S     "M173.0";
NETWORK
TITLE =
      A     "T0";
      A(;
      ON    "MAP_DI".DB91_DBX061_6;
      O     "M173.0";
      );
      A     "M188.0";
      =     "Db Plc <=> HMI".CAGE12_1.DB100_DBX128_00;
NETWORK
TITLE = CAGE 12 PRESENCE OF MAN
      A     "T0";
      AN    "MAP_DI".DB91_DBX061_7;
      AN    "M180.1";
      A     "M188.0";
      =     "Db Plc <=> HMI".CAGE12_1.DB100_DBX128_01;
NETWORK
TITLE = CAGE 12 LOADING ENGAGED
      A     "T0";
      A     "MAP_DI".DB91_DBX060_5;
      AN    "MAP_DI".DB91_DBX060_6;
      A     "M15.2";
      =     "Db Plc <=> HMI".CAGE12_1.DB100_DBX128_02;
NETWORK
TITLE = CAGE 12 LOADING GEAR BOX NOT ENGAGED
      A     "T0";
      AN    "MAP_DI".DB91_DBX060_5;
      AN    "MAP_DI".DB91_DBX060_6;
      =     "Db Plc <=> HMI".CAGE12_1.DB100_DBX128_03;
NETWORK
TITLE = CAGE 12 LOADING MOTOR OVERLOAD
      A     "T0";
      A     "MAP_DI".DB91_DBX058_2;
      =     "Db Plc <=> HMI".CAGE12_1.DB100_DBX128_06;
NETWORK
TITLE = CAGE 12 AIR PIPE NOT IN POSITION
      A     "T0";
      A     "M180.1";
      AN    "MAP_DI".DB91_DBX060_7;
      A     "M188.0";
      S     "M170.7";
NETWORK
TITLE =
      A     "T0";
      A(;
      ON    "MAP_DI".DB91_DBX060_7;
      O     "M170.7";
      );
      =     "Db Plc <=> HMI".CAGE12_1.DB100_DBX128_05;
NETWORK
TITLE = CAGE 12 PISTON INSIDE CAGE
      A     "T0";
      A     "M180.1";
      AN    "MAP_DI".DB91_DBX060_4;
      A     "M188.0";
      S     "M171.0";
NETWORK
TITLE =
      A     "T0";
      A(;
      ON    "MAP_DI".DB91_DBX060_4;
      O     "M171.0";
      );
      =     "Db Plc <=> HMI".CAGE12_1.DB100_DBX128_07;
NETWORK
TITLE = CAGE 12 24VDC POWER SUPPLY OVERLOAD
      A     "T0";
      AN    "MAP_DI".DB91_DBX058_1;
      =     "Db Plc <=> HMI".CAGE12_1.DB100_DBX129_00;
NETWORK
TITLE = CAGE 12 230VAC POWER SUPPLY OVERLOAD
      A     "T0";
      AN    "MAP_DI".DB91_DBX058_0;
      =     "Db Plc <=> HMI".CAGE12_1.DB100_DBX129_01;
NETWORK
TITLE = CAGE 12 MOTOR BLOWER OVERLOAD
      A     "T0";
      A     "MAP_DI".DB91_DBX058_3;
      =     "Db Plc <=> HMI".CAGE12_1.DB100_DBX129_02;
NETWORK
TITLE = CAGE 12 LOADING PLATFORM MOTOR OVERLOAD
NETWORK
TITLE = CAGE 12 GUARD BLOWER MOTOR OVERLOAD
      A     "T0";
      A     "MAP_DI".DB91_DBX058_7;
      =     "Db Plc <=> HMI".CAGE12_1.DB100_DBX129_05;
NETWORK
TITLE = CAGE 12 OPEN FRONT DOOR
//      U(    
//      U(    
//      U     T      0
//      U     M    178.0
//      O     M    180.1
//      O     M     21.3
//      )     
//      L     S5T#2S
//      SE    T     35
//      NOP   0
//      NOP   0
//      NOP   0
//      U     T     35
//      )     
//      UN    DB91.DBX   61.3
//      U     M    188.0
//      S     DB100.DBX  129.6
NETWORK
TITLE = CAGE 12 OPEN REAR DOORS
      A     "T0";
      A     "M180.1";
      AN    "MAP_DI".DB91_DBX061_4;
      A     "M188.0";
      S     "M172.5";
NETWORK
TITLE =
      A     "T0";
      A(;
      ON    "MAP_DI".DB91_DBX061_4;
      O     "M172.5";
      );
      A     "M188.0";
      =     "Db Plc <=> HMI".CAGE12_1.DB100_DBX129_07;
NETWORK
TITLE = CAGE 12 BREAK WIRE FROM RING 
      A     "T0";
      A     "T1";
      AN    "MAP_DI".DB91_DBX061_2;
      A     "M188.0";
      S     "Db Plc <=> HMI".Cage12_3.DB100_DBX133_06;
NETWORK
TITLE = CAGE 12 MAIN AIR MINIMUM PRESSURE
      A     "T0";
      A     "M180.1";
      AN    "MAP_DI".DB91_DBX060_2;
      A     "M188.0";
      S     "M172.3";
NETWORK
TITLE =
      A     "T0";
      A(;
      ON    "MAP_DI".DB91_DBX060_2;
      O     "M172.3";
      );
      =     "Db Plc <=> HMI".Cage12_4.DB100_DBX134_00;
NETWORK
TITLE = CAGE 12 BOBBIN BRAKES AIR TANK MINIMUM PRESSURE
      A     "T0";
      AN    "Db Plc <=> HMI".PROFIBUS.DB100_DBX100_7;
      AN    "MAP_DI".DB91_DBX067_0;
      A     "M188.0";
      S     "Db Plc <=> HMI".Cage12_4.DB100_DBX134_01;
NETWORK
TITLE = CAGE 12 LINE 1 PINTLES OPEN
      A     "T0";
      A     "M180.1";
      AN    "MAP_DI".DB91_DBX067_1;
      A     "M188.0";
      S     "M171.1";
NETWORK
TITLE =
      A     "T0";
      A(;
      ON    "MAP_DI".DB91_DBX067_1;
      O     "M171.1";
      );
      =     "Db Plc <=> HMI".Cage12_4.DB100_DBX134_02;
NETWORK
TITLE = CAGE 12 LINE 2 PINTLES OPEN
      A     "T0";
      A     "M180.1";
      AN    "MAP_DI".DB91_DBX067_2;
      A     "M188.0";
      S     "M171.2";
NETWORK
TITLE =
      A     "T0";
      A(;
      ON    "MAP_DI".DB91_DBX067_2;
      O     "M171.2";
      );
      =     "Db Plc <=> HMI".Cage12_4.DB100_DBX134_03;
NETWORK
TITLE = CAGE 12 LINE 3 PINTLES OPEN
      A     "T0";
      A     "M180.1";
      AN    "MAP_DI".DB91_DBX067_3;
      A     "M188.0";
      S     "M171.3";
NETWORK
TITLE =
      A     "T0";
      A(;
      ON    "MAP_DI".DB91_DBX067_3;
      O     "M171.3";
      );
      =     "Db Plc <=> HMI".Cage12_4.DB100_DBX134_04;
NETWORK
TITLE = CAGE 12 OPEN PINTLES LAMP
      ON    "MAP_DI".DB91_DBX067_1;
      ON    "MAP_DI".DB91_DBX067_2;
      ON    "MAP_DI".DB91_DBX067_3;
      =     "M179.3";
      =     "MAP_DO".DB93_DBX042_0;
NETWORK
TITLE = CAGE 12 MOTOR DRIVE FAULT
      A     "T0";
      A     "Drives --> Plc".CAGE_12_STATUS_W1.DB1_DBX321_3;
      S     "Db Plc <=> HMI".Cage12_4.DB100_DBX134_05;
NETWORK
TITLE = CAGE 12 MOTOR OVERTEMPERATURE
      A     "T0";
      A     "Drives --> Plc".CAGE_12_STATUS_W2.DB1_DBX322_1;
      S     "Db Plc <=> HMI".Cage12_4.DB100_DBX134_06;
NETWORK
TITLE = CAGE 12 OVERSPEED
      A     "T0";
      A     "M180.1";
      A(;
      L     "Cage 12".DB25_DBD108;
      L     3.250000e+02;
      >=R;
      );
      A     "M188.0";
      S     "Db Plc <=> HMI".Cage12_4.DB100_DBX134_07;
NETWORK
TITLE = CAGE 12 BRAKES CONTROL
      A     "T0";
      A     "T2";
      AN    "MAP_DI".DB91_DBX060_1;
      A     "M188.0";
      S     "Db Plc <=> HMI".Cage12_4.DB100_DBX135_00;
NETWORK
TITLE = CAGE 12 PLATFORM UP
NETWORK
TITLE = CAGE 12 HYDRAULIC UNIT MINIMUM OIL LEVEL  
NETWORK
TITLE = CAGE 12 GENERAL ALARM
      AN    "Db Plc <=> HMI".PROFIBUS.DB100_DBX100_2;
      AN    "Db Plc <=> HMI".PROFIBUS.DB100_DBX100_7;
      AN    "Db Plc <=> HMI".CAGE12_1.DB100_DBX128_00;
      AN    "Db Plc <=> HMI".CAGE12_1.DB100_DBX128_01;
      AN    "Db Plc <=> HMI".CAGE12_1.DB100_DBX128_03;
      AN    "Db Plc <=> HMI".CAGE12_1.DB100_DBX128_04;
      AN    "Db Plc <=> HMI".CAGE12_1.DB100_DBX128_05;
      AN    "Db Plc <=> HMI".CAGE12_1.DB100_DBX128_07;
      AN    "Db Plc <=> HMI".CAGE12_1.DB100_DBX129_00;
      AN    "Db Plc <=> HMI".CAGE12_1.DB100_DBX129_01;
      AN    "Db Plc <=> HMI".CAGE12_1.DB100_DBX129_02;
      AN    "Db Plc <=> HMI".CAGE12_1.DB100_DBX129_06;
      AN    "Db Plc <=> HMI".CAGE12_1.DB100_DBX129_07;
      AN    "Db Plc <=> HMI".Cage12_2.DB100_DBX130_00;
      AN    "Db Plc <=> HMI".Cage12_2.DB100_DBX130_01;
      AN    "Db Plc <=> HMI".Cage12_2.DB100_DBX130_02;
      AN    "Db Plc <=> HMI".Cage12_2.DB100_DBX130_03;
      AN    "Db Plc <=> HMI".Cage12_2.DB100_DBX130_04;
      AN    "Db Plc <=> HMI".Cage12_2.DB100_DBX130_05;
      AN    "Db Plc <=> HMI".Cage12_2.DB100_DBX130_06;
      AN    "Db Plc <=> HMI".Cage12_2.DB100_DBX130_07;
      AN    "Db Plc <=> HMI".Cage12_2.DB100_DBX131_00;
      AN    "Db Plc <=> HMI".Cage12_2.DB100_DBX131_01;
      AN    "Db Plc <=> HMI".Cage12_2.DB100_DBX131_02;
      AN    "Db Plc <=> HMI".Cage12_2.DB100_DBX131_03;
      AN    "Db Plc <=> HMI".Cage12_3.DB100_DBX133_06;
      AN    "Db Plc <=> HMI".Cage12_3.DB100_DBX133_07;
      AN    "Db Plc <=> HMI".Cage12_4.DB100_DBX134_00;
      AN    "Db Plc <=> HMI".Cage12_4.DB100_DBX134_01;
      AN    "Db Plc <=> HMI".Cage12_4.DB100_DBX134_02;
      AN    "Db Plc <=> HMI".Cage12_4.DB100_DBX134_03;
      AN    "Db Plc <=> HMI".Cage12_4.DB100_DBX134_04;
      AN    "Db Plc <=> HMI".Cage12_4.DB100_DBX134_05;
      AN    "Db Plc <=> HMI".Cage12_4.DB100_DBX134_06;
      AN    "Db Plc <=> HMI".Cage12_4.DB100_DBX134_07;
      AN    "Db Plc <=> HMI".Cage12_4.DB100_DBX135_00;
      ON    "M188.0";
      =     "M195.7";
END_FUNCTION

